SPLINE
SPL {X  -136.508, Y  +299.059, Z    +0.000, E1  +318.212, E3 -183209.129}
SPL {X  -153.176, Y  +336.305, Z    +0.000, E1  +330.872, E3 -183235.694}
SPL {X  -158.263, Y  +359.056, Z    +0.000, E1  +342.551, E3 -183242.369}
SPL {X  -159.616, Y  +371.564, Z    +0.000, E1  +350.434, E3 -183244.274}
SPL {X  -159.983, Y  +381.031, Z    +0.000, E1  +357.053, E3 -183244.964}
SPL {X  -159.990, Y  +384.524, Z    +0.000, E1  +359.995, E3 -183245.052}
SPL {X  -159.990, Y  +386.890, Z    +0.000, E1  +362.742, E3 -183245.108}
SPL {X  -159.990, Y  +392.248, Z    +0.000, E1  +370.895, E3 -183245.436}
SPL {X  -159.990, Y  +398.030, Z    +0.000, E1  +380.706, E3 -183246.087}
SPL {X  -159.990, Y  +404.858, Z    +0.000, E1  +391.125, E3 -183247.331}
SPL {X  -159.990, Y  +416.328, Z    +0.000, E1  +404.105, E3 -183250.268}
SPL {X  -159.990, Y  +459.824, Z    +0.000, E1  +420.326, E3 -183270.190}
SPL {X  -159.990, Y  +565.974, Z    +0.000, E1  +423.959, E3 -183353.679}
SPL {X  -159.990, Y  +578.588, Z    +0.000, E1  +423.918, E3 -183366.858}
SPL {X  -159.990, Y  +590.041, Z    +0.000, E1  +423.939, E3 -183378.713}
SPL {X  -159.990, Y  +601.352, Z    +0.000, E1  +423.918, E3 -183390.500}
SPL {X  -159.990, Y  +610.973, Z    +0.000, E1  +423.927, E3 -183400.468}
SPL {X  -159.990, Y  +624.756, Z    +0.000, E1  +423.949, E3 -183414.746}
SPL {X  -159.990, Y  +640.674, Z    +0.000, E1  +423.943, E3 -183431.282}
SPL {X  -159.990, Y  +652.355, Z    +0.000, E1  +423.915, E3 -183443.481}
SPL {X  -159.990, Y  +665.748, Z    +0.000, E1  +423.953, E3 -183457.335}
SPL {X  -159.643, Y  +682.032, Z    +0.000, E1  +423.894, E3 -183474.628}
SPL {X  -158.070, Y  +696.212, Z    +0.000, E1  +423.682, E3 -183490.966}
SPL {X  -155.481, Y  +709.215, Z    +0.000, E1  +423.310, E3 -183507.157}
SPL {X  -153.138, Y  +717.820, Z    +0.000, E1  +422.909, E3 -183518.576}
SPL {X  -151.229, Y  +723.716, Z    +0.000, E1  +422.630, E3 -183526.585}
SPL {X  -149.219, Y  +729.211, Z    +0.000, E1  +422.307, E3 -183534.294}
SPL {X  -146.537, Y  +735.716, Z    +0.000, E1  +421.906, E3 -183543.637}
SPL {X  -143.476, Y  +742.291, Z    +0.000, E1  +421.379, E3 -183553.397}
SPL {X  -141.015, Y  +747.074, Z    +0.000, E1  +420.958, E3 -183560.653}
SPL {X  -137.271, Y  +753.679, Z    +0.000, E1  +420.346, E3 -183570.791}
SPL {X  -133.306, Y  +759.967, Z    +0.000, E1  +419.584, E3 -183580.743}
SPL {X  -112.019, Y  +785.730, Z    +0.000, E1  +410.795, E3 -183683.484}
ENDSPLINE

SPLINE
SPL {X  -138.335, Y  +751.876, Z    +0.000, E1  +401.001, E3 -183797.783}
SPL {X  -150.285, Y  +726.376, Z    +0.000, E1  +392.667, E3 -183816.192}
SPL {X  -156.272, Y  +705.789, Z    +0.000, E1  +383.396, E3 -183823.828}
SPL {X  -159.413, Y  +685.076, Z    +0.000, E1  +371.341, E3 -183827.966}
SPL {X  -159.964, Y  +674.389, Z    +0.000, E1  +363.956, E3 -183828.937}
SPL {X  -159.990, Y  +670.214, Z    +0.000, E1  +360.653, E3 -183829.083}
SPL {X  -159.990, Y  +669.154, Z    +0.000, E1  +359.694, E3 -183829.092}
SPL {X  -159.990, Y  +666.004, Z    +0.000, E1  +355.742, E3 -183829.192}
SPL {X  -159.990, Y  +661.286, Z    +0.000, E1  +348.294, E3 -183829.508}
SPL {X  -159.990, Y  +656.470, Z    +0.000, E1  +340.220, E3 -183830.046}
SPL {X  -159.990, Y  +651.555, Z    +0.000, E1  +332.416, E3 -183830.854}
SPL {X  -159.990, Y  +640.109, Z    +0.000, E1  +318.471, E3 -183833.683}
SPL {X  -159.990, Y  +589.014, Z    +0.000, E1  +298.500, E3 -183855.548}
SPL {X  -159.990, Y  +484.717, Z    +0.000, E1  +295.169, E3 -183933.731}
SPL {X  -159.990, Y  +469.712, Z    +0.000, E1  +295.152, E3 -183948.668}
SPL {X  -159.990, Y  +456.089, Z    +0.000, E1  +295.174, E3 -183962.284}
SPL {X  -159.990, Y  +443.816, Z    +0.000, E1  +295.158, E3 -183974.484}
SPL {X  -159.990, Y  +405.035, Z    +0.000, E1  +292.209, E3 -183986.755}
SPL {X  -159.990, Y  +397.824, Z    +0.000, E1  +292.709, E3 -183997.117}
SPL {X  -159.990, Y  +393.786, Z    +0.000, E1  +293.391, E3 -184006.436}
SPL {X  -159.990, Y  +385.177, Z    +0.000, E1  +294.011, E3 -184019.553}
SPL {X  -159.935, Y  +378.300, Z    +0.000, E1  +295.100, E3 -184034.762}
SPL {X  -159.716, Y  +373.142, Z    +0.000, E1  +296.084, E3 -184047.303}
SPL {X  -158.852, Y  +363.449, Z    +0.000, E1  +296.568, E3 -184061.253}
SPL {X  -157.299, Y  +353.279, Z    +0.000, E1  +296.835, E3 -184073.685}
SPL {X  -155.242, Y  +343.812, Z    +0.000, E1  +297.102, E3 -184085.733}
SPL {X  -151.999, Y  +332.569, Z    +0.000, E1  +297.592, E3 -184100.891}
SPL {X  -148.909, Y  +323.994, Z    +0.000, E1  +298.107, E3 -184113.064}
SPL {X  -146.667, Y  +318.581, Z    +0.000, E1  +298.485, E3 -184120.985}
SPL {X  -144.416, Y  +313.647, Z    +0.000, E1  +298.845, E3 -184128.321}
SPL {X  -141.484, Y  +307.808, Z    +0.000, E1  +299.342, E3 -184137.214}
SPL {X  -139.055, Y  +303.377, Z    +0.000, E1  +299.788, E3 -184144.126}
SPL {X  -136.464, Y  +298.988, Z    +0.000, E1  +300.231, E3 -184151.001}
SPL {X  -133.486, Y  +294.305, Z    +0.000, E1  +300.785, E3 -184158.463}
SPL {X  -111.268, Y  +267.538, Z    +0.000, E1  +309.436, E3 -184266.362}
ENDSPLINE

SPLINE
SPL {X  -140.331, Y  +305.662, Z    +0.000, E1  +319.927, E3 -184378.430}
SPL {X  -153.176, Y  +336.305, Z    +0.000, E1  +330.872, E3 -184396.984}
SPL {X  -158.263, Y  +359.056, Z    +0.000, E1  +342.551, E3 -184403.659}
SPL {X  -159.616, Y  +371.564, Z    +0.000, E1  +350.434, E3 -184405.564}
SPL {X  -159.946, Y  +378.747, Z    +0.000, E1  +355.440, E3 -184406.159}
SPL {X  -159.990, Y  +384.172, Z    +0.000, E1  +359.586, E3 -184406.337}
SPL {X  -159.990, Y  +385.853, Z    +0.000, E1  +361.539, E3 -184406.362}
SPL {X  -159.990, Y  +389.234, Z    +0.000, E1  +366.142, E3 -184406.507}
SPL {X  -159.990, Y  +395.814, Z    +0.000, E1  +376.762, E3 -184407.108}
SPL {X  -159.990, Y  +404.858, Z    +0.000, E1  +391.125, E3 -184408.622}
SPL {X  -159.990, Y  +416.328, Z    +0.000, E1  +404.105, E3 -184411.559}
SPL {X  -159.990, Y  +459.824, Z    +0.000, E1  +420.326, E3 -184431.481}
SPL {X  -159.990, Y  +565.974, Z    +0.000, E1  +423.959, E3 -184514.969}
SPL {X  -159.990, Y  +578.588, Z    +0.000, E1  +423.918, E3 -184528.149}
SPL {X  -159.990, Y  +590.041, Z    +0.000, E1  +423.939, E3 -184540.004}
SPL {X  -159.990, Y  +601.352, Z    +0.000, E1  +423.918, E3 -184551.790}
SPL {X  -159.990, Y  +610.973, Z    +0.000, E1  +423.927, E3 -184561.758}
SPL {X  -159.990, Y  +624.756, Z    +0.000, E1  +423.949, E3 -184576.036}
SPL {X  -159.990, Y  +636.914, Z    +0.000, E1  +423.917, E3 -184588.712}
SPL {X  -159.990, Y  +648.849, Z    +0.000, E1  +423.945, E3 -184601.069}
SPL {X  -159.990, Y  +661.195, Z    +0.000, E1  +423.915, E3 -184613.970}
SPL {X  -159.965, Y  +674.349, Z    +0.000, E1  +423.939, E3 -184627.607}
SPL {X  -159.404, Y  +685.179, Z    +0.000, E1  +423.831, E3 -184639.486}
SPL {X  -158.535, Y  +693.032, Z    +0.000, E1  +423.713, E3 -184648.535}
SPL {X  -156.949, Y  +702.544, Z    +0.000, E1  +423.501, E3 -184660.041}
SPL {X  -154.903, Y  +711.525, Z    +0.000, E1  +423.186, E3 -184671.512}
SPL {X  -153.138, Y  +717.820, Z    +0.000, E1  +422.909, E3 -184679.866}
SPL {X  -151.229, Y  +723.716, Z    +0.000, E1  +422.630, E3 -184687.876}
SPL {X  -149.219, Y  +729.211, Z    +0.000, E1  +422.307, E3 -184695.584}
SPL {X  -146.537, Y  +735.716, Z    +0.000, E1  +421.906, E3 -184704.927}
SPL {X  -143.476, Y  +742.291, Z    +0.000, E1  +421.379, E3 -184714.687}
SPL {X  -141.015, Y  +747.074, Z    +0.000, E1  +420.958, E3 -184721.943}
SPL {X  -137.271, Y  +753.679, Z    +0.000, E1  +420.346, E3 -184732.082}
SPL {X  -133.306, Y  +759.967, Z    +0.000, E1  +419.584, E3 -184742.033}
SPL {X  -112.019, Y  +785.730, Z    +0.000, E1  +410.795, E3 -184844.774}
ENDSPLINE

SPLINE
SPL {X  -138.335, Y  +751.876, Z    +0.000, E1  +401.001, E3 -184959.073}
SPL {X  -150.285, Y  +726.376, Z    +0.000, E1  +392.667, E3 -184977.482}
SPL {X  -156.272, Y  +705.789, Z    +0.000, E1  +383.396, E3 -184985.118}
SPL {X  -159.413, Y  +685.076, Z    +0.000, E1  +371.341, E3 -184989.257}
SPL {X  -159.964, Y  +674.389, Z    +0.000, E1  +363.956, E3 -184990.227}
SPL {X  -159.990, Y  +669.409, Z    +0.000, E1  +360.015, E3 -184990.381}
SPL {X  -159.990, Y  +667.272, Z    +0.000, E1  +357.329, E3 -184990.424}
SPL {X  -159.990, Y  +664.817, Z    +0.000, E1  +353.836, E3 -184990.537}
SPL {X  -159.990, Y  +661.286, Z    +0.000, E1  +348.294, E3 -184990.799}
SPL {X  -159.990, Y  +654.198, Z    +0.000, E1  +336.753, E3 -184991.710}
SPL {X  -159.990, Y  +640.109, Z    +0.000, E1  +318.471, E3 -184994.973}
SPL {X  -159.990, Y  +589.014, Z    +0.000, E1  +298.500, E3 -185016.838}
SPL {X  -159.990, Y  +484.717, Z    +0.000, E1  +295.169, E3 -185095.022}
SPL {X  -159.990, Y  +474.300, Z    +0.000, E1  +295.184, E3 -185105.449}
SPL {X  -159.990, Y  +465.825, Z    +0.000, E1  +295.182, E3 -185113.889}
SPL {X  -159.990, Y  +451.559, Z    +0.000, E1  +295.138, E3 -185128.026}
SPL {X  -159.990, Y  +438.393, Z    +0.000, E1  +295.184, E3 -185141.248}
SPL {X  -159.990, Y  +405.035, Z    +0.000, E1  +292.209, E3 -185148.045}
SPL {X  -159.990, Y  +395.217, Z    +0.000, E1  +293.078, E3 -185164.154}
SPL {X  -159.990, Y  +387.038, Z    +0.000, E1  +293.844, E3 -185177.582}
SPL {X  -159.983, Y  +380.995, Z    +0.000, E1  +294.559, E3 -185189.151}
SPL {X  -159.795, Y  +374.602, Z    +0.000, E1  +295.796, E3 -185205.170}
SPL {X  -158.852, Y  +363.449, Z    +0.000, E1  +296.568, E3 -185222.543}
SPL {X  -156.653, Y  +349.995, Z    +0.000, E1  +296.892, E3 -185239.047}
SPL {X  -153.792, Y  +338.401, Z    +0.000, E1  +297.323, E3 -185254.216}
SPL {X  -151.244, Y  +330.327, Z    +0.000, E1  +297.748, E3 -185265.369}
SPL {X  -148.909, Y  +323.994, Z    +0.000, E1  +298.107, E3 -185274.355}
SPL {X  -146.667, Y  +318.581, Z    +0.000, E1  +298.485, E3 -185282.275}
SPL {X  -144.416, Y  +313.647, Z    +0.000, E1  +298.845, E3 -185289.611}
SPL {X  -141.484, Y  +307.808, Z    +0.000, E1  +299.342, E3 -185298.504}
SPL {X  -139.055, Y  +303.377, Z    +0.000, E1  +299.788, E3 -185305.417}
SPL {X  -136.464, Y  +298.988, Z    +0.000, E1  +300.231, E3 -185312.291}
SPL {X  -133.486, Y  +294.305, Z    +0.000, E1  +300.785, E3 -185319.753}
SPL {X  -111.268, Y  +267.538, Z    +0.000, E1  +309.436, E3 -185427.652}
ENDSPLINE

SPLINE
SPL {X  -140.331, Y  +305.662, Z    +0.000, E1  +319.927, E3 -185539.720}
SPL {X  -153.176, Y  +336.305, Z    +0.000, E1  +330.872, E3 -185558.275}
SPL {X  -157.724, Y  +355.668, Z    +0.000, E1  +340.639, E3 -185564.283}
SPL {X  -159.465, Y  +369.545, Z    +0.000, E1  +349.053, E3 -185566.605}
SPL {X  -159.983, Y  +381.031, Z    +0.000, E1  +357.053, E3 -185567.545}
SPL {X  -159.990, Y  +384.524, Z    +0.000, E1  +359.995, E3 -185567.633}
SPL {X  -159.990, Y  +386.890, Z    +0.000, E1  +362.742, E3 -185567.689}
SPL {X  -159.990, Y  +392.248, Z    +0.000, E1  +370.895, E3 -185568.016}
SPL {X  -159.990, Y  +398.030, Z    +0.000, E1  +380.706, E3 -185568.668}
SPL {X  -159.990, Y  +404.858, Z    +0.000, E1  +391.125, E3 -185569.912}
SPL {X  -159.990, Y  +416.328, Z    +0.000, E1  +404.105, E3 -185572.849}
SPL {X  -159.990, Y  +459.824, Z    +0.000, E1  +420.326, E3 -185592.771}
SPL {X  -159.990, Y  +565.974, Z    +0.000, E1  +423.959, E3 -185676.260}
SPL {X  -159.990, Y  +578.588, Z    +0.000, E1  +423.918, E3 -185689.439}
SPL {X  -159.990, Y  +590.041, Z    +0.000, E1  +423.939, E3 -185701.294}
SPL {X  -159.990, Y  +601.352, Z    +0.000, E1  +423.918, E3 -185713.080}
SPL {X  -159.990, Y  +614.998, Z    +0.000, E1  +423.962, E3 -185727.165}
SPL {X  -159.990, Y  +628.256, Z    +0.000, E1  +423.919, E3 -185741.014}
SPL {X  -159.990, Y  +640.674, Z    +0.000, E1  +423.943, E3 -185753.863}
SPL {X  -159.990, Y  +657.298, Z    +0.000, E1  +423.953, E3 -185771.135}
SPL {X  -159.990, Y  +670.369, Z    +0.000, E1  +423.912, E3 -185784.793}
SPL {X  -159.643, Y  +682.032, Z    +0.000, E1  +423.894, E3 -185797.208}
SPL {X  -158.070, Y  +696.212, Z    +0.000, E1  +423.682, E3 -185813.547}
SPL {X  -155.481, Y  +709.215, Z    +0.000, E1  +423.310, E3 -185829.738}
SPL {X  -153.138, Y  +717.820, Z    +0.000, E1  +422.909, E3 -185841.156}
SPL {X  -151.229, Y  +723.716, Z    +0.000, E1  +422.630, E3 -185849.166}
SPL {X  -149.219, Y  +729.211, Z    +0.000, E1  +422.307, E3 -185856.874}
SPL {X  -146.537, Y  +735.716, Z    +0.000, E1  +421.906, E3 -185866.217}
SPL {X  -143.476, Y  +742.291, Z    +0.000, E1  +421.379, E3 -185875.977}
SPL {X  -141.015, Y  +747.074, Z    +0.000, E1  +420.958, E3 -185883.234}
SPL {X  -137.271, Y  +753.679, Z    +0.000, E1  +420.346, E3 -185893.372}
SPL {X  -133.306, Y  +759.967, Z    +0.000, E1  +419.584, E3 -185903.324}
SPL {X  -112.019, Y  +785.730, Z    +0.000, E1  +410.795, E3 -186006.065}
ENDSPLINE

SPLINE
SPL {X  -126.527, Y  +769.417, Z    +0.000, E1  +405.012, E3 -186095.917}
SPL {X  -141.954, Y  +745.296, Z    +0.000, E1  +399.179, E3 -186127.115}
SPL {X  -153.384, Y  +716.997, Z    +0.000, E1  +388.774, E3 -186142.735}
SPL {X  -158.303, Y  +694.673, Z    +0.000, E1  +377.238, E3 -186149.046}
SPL {X  -159.604, Y  +682.609, Z    +0.000, E1  +369.664, E3 -186150.856}
SPL {X  -159.964, Y  +674.389, Z    +0.000, E1  +363.956, E3 -186151.518}
SPL {X  -159.990, Y  +669.409, Z    +0.000, E1  +360.015, E3 -186151.671}
SPL {X  -159.990, Y  +666.004, Z    +0.000, E1  +355.742, E3 -186151.773}
SPL {X  -159.990, Y  +661.286, Z    +0.000, E1  +348.294, E3 -186152.089}
SPL {X  -159.990, Y  +654.198, Z    +0.000, E1  +336.753, E3 -186153.000}
SPL {X  -159.990, Y  +640.109, Z    +0.000, E1  +318.471, E3 -186156.263}
SPL {X  -159.990, Y  +589.014, Z    +0.000, E1  +298.500, E3 -186178.129}
SPL {X  -159.990, Y  +484.717, Z    +0.000, E1  +295.169, E3 -186256.312}
SPL {X  -159.990, Y  +474.300, Z    +0.000, E1  +295.184, E3 -186266.740}
SPL {X  -159.990, Y  +465.825, Z    +0.000, E1  +295.182, E3 -186275.179}
SPL {X  -159.990, Y  +451.559, Z    +0.000, E1  +295.138, E3 -186289.316}
SPL {X  -159.990, Y  +423.512, Z    +0.000, E1  +293.559, E3 -186303.750}
SPL {X  -159.990, Y  +399.563, Z    +0.000, E1  +292.427, E3 -186316.028}
SPL {X  -159.990, Y  +393.786, Z    +0.000, E1  +293.391, E3 -186329.017}
SPL {X  -159.990, Y  +387.038, Z    +0.000, E1  +293.844, E3 -186338.873}
SPL {X  -159.983, Y  +380.995, Z    +0.000, E1  +294.559, E3 -186350.441}
SPL {X  -159.898, Y  +377.064, Z    +0.000, E1  +295.481, E3 -186361.255}
SPL {X  -159.716, Y  +373.142, Z    +0.000, E1  +296.084, E3 -186369.884}
SPL {X  -158.852, Y  +363.449, Z    +0.000, E1  +296.568, E3 -186383.834}
SPL {X  -157.299, Y  +353.279, Z    +0.000, E1  +296.835, E3 -186396.265}
SPL {X  -155.242, Y  +343.812, Z    +0.000, E1  +297.102, E3 -186408.313}
SPL {X  -151.999, Y  +332.569, Z    +0.000, E1  +297.592, E3 -186423.472}
SPL {X  -148.909, Y  +323.994, Z    +0.000, E1  +298.107, E3 -186435.645}
SPL {X  -146.667, Y  +318.581, Z    +0.000, E1  +298.485, E3 -186443.565}
SPL {X  -144.416, Y  +313.647, Z    +0.000, E1  +298.845, E3 -186450.902}
SPL {X  -141.484, Y  +307.808, Z    +0.000, E1  +299.342, E3 -186459.795}
SPL {X  -139.055, Y  +303.377, Z    +0.000, E1  +299.788, E3 -186466.707}
SPL {X  -136.464, Y  +298.988, Z    +0.000, E1  +300.231, E3 -186473.581}
SPL {X  -133.486, Y  +294.305, Z    +0.000, E1  +300.785, E3 -186481.043}
SPL {X  -111.268, Y  +267.538, Z    +0.000, E1  +309.436, E3 -186588.942}
ENDSPLINE

SPLINE
SPL {X  -140.331, Y  +305.662, Z    +0.000, E1  +319.927, E3 -186701.011}
SPL {X  -153.176, Y  +336.305, Z    +0.000, E1  +330.872, E3 -186719.565}
SPL {X  -158.263, Y  +359.056, Z    +0.000, E1  +342.551, E3 -186726.240}
SPL {X  -159.616, Y  +371.564, Z    +0.000, E1  +350.434, E3 -186728.145}
SPL {X  -159.983, Y  +381.031, Z    +0.000, E1  +357.053, E3 -186728.835}
SPL {X  -159.990, Y  +385.049, Z    +0.000, E1  +360.437, E3 -186728.931}
SPL {X  -159.990, Y  +389.234, Z    +0.000, E1  +366.142, E3 -186729.087}
SPL {X  -159.990, Y  +395.814, Z    +0.000, E1  +376.762, E3 -186729.689}
SPL {X  -159.990, Y  +404.858, Z    +0.000, E1  +391.125, E3 -186731.202}
SPL {X  -159.990, Y  +416.328, Z    +0.000, E1  +404.105, E3 -186734.139}
SPL {X  -159.990, Y  +459.824, Z    +0.000, E1  +420.326, E3 -186754.061}
SPL {X  -159.990, Y  +565.974, Z    +0.000, E1  +423.959, E3 -186837.550}
SPL {X  -159.990, Y  +582.903, Z    +0.000, E1  +423.951, E3 -186855.147}
SPL {X  -159.990, Y  +598.374, Z    +0.000, E1  +423.941, E3 -186871.234}
SPL {X  -159.990, Y  +614.998, Z    +0.000, E1  +423.962, E3 -186888.455}
SPL {X  -159.990, Y  +632.576, Z    +0.000, E1  +423.953, E3 -186906.721}
SPL {X  -159.990, Y  +648.849, Z    +0.000, E1  +423.945, E3 -186923.650}
SPL {X  -159.990, Y  +665.748, Z    +0.000, E1  +423.953, E3 -186941.206}
SPL {X  -159.643, Y  +682.032, Z    +0.000, E1  +423.894, E3 -186958.499}
SPL {X  -158.070, Y  +696.212, Z    +0.000, E1  +423.682, E3 -186974.837}
SPL {X  -155.481, Y  +709.215, Z    +0.000, E1  +423.310, E3 -186991.028}
SPL {X  -153.138, Y  +717.820, Z    +0.000, E1  +422.909, E3 -187002.447}
SPL {X  -151.229, Y  +723.716, Z    +0.000, E1  +422.630, E3 -187010.456}
SPL {X  -148.422, Y  +731.231, Z    +0.000, E1  +422.207, E3 -187021.014}
SPL {X  -145.802, Y  +737.367, Z    +0.000, E1  +421.758, E3 -187029.967}
SPL {X  -143.476, Y  +742.291, Z    +0.000, E1  +421.379, E3 -187037.268}
SPL {X  -141.015, Y  +747.074, Z    +0.000, E1  +420.958, E3 -187044.524}
SPL {X  -138.539, Y  +751.523, Z    +0.000, E1  +420.526, E3 -187051.359}
SPL {X  -136.299, Y  +755.281, Z    +0.000, E1  +420.128, E3 -187057.220}
SPL {X  -133.306, Y  +759.967, Z    +0.000, E1  +419.584, E3 -187064.614}
SPL {X  -112.019, Y  +785.730, Z    +0.000, E1  +410.795, E3 -187167.355}
ENDSPLINE

SPLINE
SPL {X  -126.527, Y  +769.417, Z    +0.000, E1  +405.012, E3 -187257.207}
SPL {X  -141.954, Y  +745.296, Z    +0.000, E1  +399.179, E3 -187288.405}
SPL {X  -153.384, Y  +716.997, Z    +0.000, E1  +388.774, E3 -187304.025}
SPL {X  -158.303, Y  +694.673, Z    +0.000, E1  +377.238, E3 -187310.337}
SPL {X  -159.604, Y  +682.609, Z    +0.000, E1  +369.664, E3 -187312.146}
SPL {X  -159.964, Y  +674.389, Z    +0.000, E1  +363.956, E3 -187312.808}
SPL {X  -159.990, Y  +669.409, Z    +0.000, E1  +360.015, E3 -187312.961}
SPL {X  -159.990, Y  +666.004, Z    +0.000, E1  +355.742, E3 -187313.063}
SPL {X  -159.990, Y  +661.286, Z    +0.000, E1  +348.294, E3 -187313.379}
SPL {X  -159.990, Y  +654.198, Z    +0.000, E1  +336.753, E3 -187314.290}
SPL {X  -159.990, Y  +640.109, Z    +0.000, E1  +318.471, E3 -187317.554}
SPL {X  -159.990, Y  +589.014, Z    +0.000, E1  +298.500, E3 -187339.419}
SPL {X  -159.990, Y  +484.717, Z    +0.000, E1  +295.169, E3 -187417.602}
SPL {X  -159.990, Y  +469.712, Z    +0.000, E1  +295.152, E3 -187432.539}
SPL {X  -159.990, Y  +456.089, Z    +0.000, E1  +295.174, E3 -187446.155}
SPL {X  -159.990, Y  +443.816, Z    +0.000, E1  +295.158, E3 -187458.355}
SPL {X  -159.990, Y  +410.689, Z    +0.000, E1  +292.263, E3 -187466.080}
SPL {X  -159.990, Y  +399.563, Z    +0.000, E1  +292.427, E3 -187477.319}
SPL {X  -159.990, Y  +393.786, Z    +0.000, E1  +293.391, E3 -187490.307}
SPL {X  -159.990, Y  +387.038, Z    +0.000, E1  +293.844, E3 -187500.163}
SPL {X  -159.983, Y  +380.995, Z    +0.000, E1  +294.559, E3 -187511.731}
SPL {X  -159.795, Y  +374.602, Z    +0.000, E1  +295.796, E3 -187527.751}
SPL {X  -159.306, Y  +367.719, Z    +0.000, E1  +296.544, E3 -187540.208}
SPL {X  -158.431, Y  +360.219, Z    +0.000, E1  +296.670, E3 -187549.059}
SPL {X  -157.299, Y  +353.279, Z    +0.000, E1  +296.835, E3 -187557.556}
SPL {X  -156.006, Y  +347.018, Z    +0.000, E1  +297.028, E3 -187565.511}
SPL {X  -153.792, Y  +338.401, Z    +0.000, E1  +297.323, E3 -187576.797}
SPL {X  -151.244, Y  +330.327, Z    +0.000, E1  +297.748, E3 -187587.950}
SPL {X  -148.909, Y  +323.994, Z    +0.000, E1  +298.107, E3 -187596.935}
SPL {X  -146.667, Y  +318.581, Z    +0.000, E1  +298.485, E3 -187604.856}
SPL {X  -144.416, Y  +313.647, Z    +0.000, E1  +298.845, E3 -187612.192}
SPL {X  -141.484, Y  +307.808, Z    +0.000, E1  +299.342, E3 -187621.085}
SPL {X  -139.055, Y  +303.377, Z    +0.000, E1  +299.788, E3 -187627.997}
SPL {X  -136.464, Y  +298.988, Z    +0.000, E1  +300.231, E3 -187634.872}
SPL {X  -133.486, Y  +294.305, Z    +0.000, E1  +300.785, E3 -187642.334}
SPL {X  -111.268, Y  +267.538, Z    +0.000, E1  +309.436, E3 -187750.233}
ENDSPLINE

SPLINE
SPL {X  -140.331, Y  +305.662, Z    +0.000, E1  +319.927, E3 -187862.301}
SPL {X  -153.176, Y  +336.305, Z    +0.000, E1  +330.872, E3 -187880.855}
SPL {X  -158.263, Y  +359.056, Z    +0.000, E1  +342.551, E3 -187887.530}
SPL {X  -159.616, Y  +371.564, Z    +0.000, E1  +350.434, E3 -187889.435}
SPL {X  -159.983, Y  +381.031, Z    +0.000, E1  +357.053, E3 -187890.125}
SPL {X  -159.990, Y  +385.049, Z    +0.000, E1  +360.437, E3 -187890.221}
SPL {X  -159.990, Y  +389.234, Z    +0.000, E1  +366.142, E3 -187890.378}
SPL {X  -159.990, Y  +395.814, Z    +0.000, E1  +376.762, E3 -187890.979}
SPL {X  -159.990, Y  +404.858, Z    +0.000, E1  +391.125, E3 -187892.493}
SPL {X  -159.990, Y  +416.328, Z    +0.000, E1  +404.105, E3 -187895.430}
SPL {X  -159.990, Y  +459.824, Z    +0.000, E1  +420.326, E3 -187915.352}
SPL {X  -159.990, Y  +565.974, Z    +0.000, E1  +423.959, E3 -187998.840}
SPL {X  -159.990, Y  +578.588, Z    +0.000, E1  +423.918, E3 -188012.020}
SPL {X  -159.990, Y  +590.041, Z    +0.000, E1  +423.939, E3 -188023.875}
SPL {X  -159.990, Y  +601.352, Z    +0.000, E1  +423.918, E3 -188035.661}
SPL {X  -159.990, Y  +610.973, Z    +0.000, E1  +423.927, E3 -188045.629}
SPL {X  -159.990, Y  +624.756, Z    +0.000, E1  +423.949, E3 -188059.907}
SPL {X  -159.990, Y  +636.914, Z    +0.000, E1  +423.917, E3 -188072.583}
SPL {X  -159.990, Y  +648.849, Z    +0.000, E1  +423.945, E3 -188084.940}
SPL {X  -159.990, Y  +661.195, Z    +0.000, E1  +423.915, E3 -188097.841}
SPL {X  -159.965, Y  +674.349, Z    +0.000, E1  +423.939, E3 -188111.478}
SPL {X  -159.404, Y  +685.179, Z    +0.000, E1  +423.831, E3 -188123.357}
SPL {X  -158.535, Y  +693.032, Z    +0.000, E1  +423.713, E3 -188132.406}
SPL {X  -156.949, Y  +702.544, Z    +0.000, E1  +423.501, E3 -188143.912}
SPL {X  -154.903, Y  +711.525, Z    +0.000, E1  +423.186, E3 -188155.383}
SPL {X  -153.138, Y  +717.820, Z    +0.000, E1  +422.909, E3 -188163.737}
SPL {X  -151.229, Y  +723.716, Z    +0.000, E1  +422.630, E3 -188171.747}
SPL {X  -148.422, Y  +731.231, Z    +0.000, E1  +422.207, E3 -188182.304}
SPL {X  -145.802, Y  +737.367, Z    +0.000, E1  +421.758, E3 -188191.257}
SPL {X  -143.476, Y  +742.291, Z    +0.000, E1  +421.379, E3 -188198.558}
SPL {X  -141.015, Y  +747.074, Z    +0.000, E1  +420.958, E3 -188205.814}
SPL {X  -137.271, Y  +753.679, Z    +0.000, E1  +420.346, E3 -188215.953}
SPL {X  -133.306, Y  +759.967, Z    +0.000, E1  +419.584, E3 -188225.904}
SPL {X  -112.019, Y  +785.730, Z    +0.000, E1  +410.795, E3 -188328.645}
ENDSPLINE

SPLINE
SPL {X  -138.335, Y  +751.876, Z    +0.000, E1  +401.001, E3 -188442.944}
SPL {X  -150.285, Y  +726.376, Z    +0.000, E1  +392.667, E3 -188461.353}
SPL {X  -154.601, Y  +712.673, Z    +0.000, E1  +386.751, E3 -188466.958}
SPL {X  -158.303, Y  +694.673, Z    +0.000, E1  +377.238, E3 -188471.627}
SPL {X  -159.774, Y  +679.819, Z    +0.000, E1  +367.840, E3 -188473.701}
SPL {X  -159.990, Y  +671.106, Z    +0.000, E1  +361.459, E3 -188474.222}
SPL {X  -159.990, Y  +669.154, Z    +0.000, E1  +359.694, E3 -188474.254}
SPL {X  -159.990, Y  +666.004, Z    +0.000, E1  +355.742, E3 -188474.353}
SPL {X  -159.990, Y  +661.286, Z    +0.000, E1  +348.294, E3 -188474.670}
SPL {X  -159.990, Y  +654.198, Z    +0.000, E1  +336.753, E3 -188475.581}
SPL {X  -159.990, Y  +640.109, Z    +0.000, E1  +318.471, E3 -188478.844}
SPL {X  -159.990, Y  +589.014, Z    +0.000, E1  +298.500, E3 -188500.709}
SPL {X  -159.990, Y  +484.717, Z    +0.000, E1  +295.169, E3 -188578.893}
SPL {X  -159.990, Y  +469.712, Z    +0.000, E1  +295.152, E3 -188593.830}
SPL {X  -159.990, Y  +456.089, Z    +0.000, E1  +295.174, E3 -188607.445}
SPL {X  -159.990, Y  +443.816, Z    +0.000, E1  +295.158, E3 -188619.646}
SPL {X  -159.990, Y  +405.035, Z    +0.000, E1  +292.209, E3 -188631.916}
SPL {X  -159.990, Y  +395.217, Z    +0.000, E1  +293.078, E3 -188648.025}
SPL {X  -159.990, Y  +385.177, Z    +0.000, E1  +294.011, E3 -188664.714}
SPL {X  -159.935, Y  +378.300, Z    +0.000, E1  +295.100, E3 -188679.924}
SPL {X  -159.533, Y  +370.414, Z    +0.000, E1  +296.253, E3 -188696.833}
SPL {X  -158.431, Y  +360.219, Z    +0.000, E1  +296.670, E3 -188710.349}
SPL {X  -157.299, Y  +353.279, Z    +0.000, E1  +296.835, E3 -188718.846}
SPL {X  -155.242, Y  +343.812, Z    +0.000, E1  +297.102, E3 -188730.894}
SPL {X  -151.999, Y  +332.569, Z    +0.000, E1  +297.592, E3 -188746.052}
SPL {X  -148.909, Y  +323.994, Z    +0.000, E1  +298.107, E3 -188758.226}
SPL {X  -146.667, Y  +318.581, Z    +0.000, E1  +298.485, E3 -188766.146}
SPL {X  -144.416, Y  +313.647, Z    +0.000, E1  +298.845, E3 -188773.482}
SPL {X  -141.484, Y  +307.808, Z    +0.000, E1  +299.342, E3 -188782.375}
SPL {X  -139.055, Y  +303.377, Z    +0.000, E1  +299.788, E3 -188789.288}
SPL {X  -136.464, Y  +298.988, Z    +0.000, E1  +300.231, E3 -188796.162}
SPL {X  -133.486, Y  +294.305, Z    +0.000, E1  +300.785, E3 -188803.624}
SPL {X  -111.268, Y  +267.538, Z    +0.000, E1  +309.436, E3 -188911.523}
ENDSPLINE

SPLINE
SPL {X  -140.331, Y  +305.662, Z    +0.000, E1  +319.927, E3 -189023.591}
SPL {X  -153.176, Y  +336.305, Z    +0.000, E1  +330.872, E3 -189042.146}
SPL {X  -157.724, Y  +355.668, Z    +0.000, E1  +340.639, E3 -189048.154}
SPL {X  -159.465, Y  +369.545, Z    +0.000, E1  +349.053, E3 -189050.476}
SPL {X  -159.983, Y  +381.031, Z    +0.000, E1  +357.053, E3 -189051.416}
SPL {X  -159.990, Y  +384.524, Z    +0.000, E1  +359.995, E3 -189051.504}
SPL {X  -159.990, Y  +385.853, Z    +0.000, E1  +361.539, E3 -189051.523}
SPL {X  -159.990, Y  +389.234, Z    +0.000, E1  +366.142, E3 -189051.668}
SPL {X  -159.990, Y  +395.814, Z    +0.000, E1  +376.762, E3 -189052.269}
SPL {X  -159.990, Y  +404.858, Z    +0.000, E1  +391.125, E3 -189053.783}
SPL {X  -159.990, Y  +416.328, Z    +0.000, E1  +404.105, E3 -189056.720}
SPL {X  -159.990, Y  +459.824, Z    +0.000, E1  +420.326, E3 -189076.642}
SPL {X  -159.990, Y  +561.459, Z    +0.000, E1  +423.923, E3 -189155.508}
SPL {X  -159.990, Y  +574.787, Z    +0.000, E1  +423.950, E3 -189169.305}
SPL {X  -159.990, Y  +590.041, Z    +0.000, E1  +423.939, E3 -189185.165}
SPL {X  -159.990, Y  +601.352, Z    +0.000, E1  +423.918, E3 -189196.951}
SPL {X  -159.990, Y  +614.998, Z    +0.000, E1  +423.962, E3 -189211.036}
SPL {X  -159.990, Y  +628.256, Z    +0.000, E1  +423.919, E3 -189224.885}
SPL {X  -159.990, Y  +640.674, Z    +0.000, E1  +423.943, E3 -189237.734}
SPL {X  -159.990, Y  +657.298, Z    +0.000, E1  +423.953, E3 -189255.006}
SPL {X  -159.990, Y  +670.369, Z    +0.000, E1  +423.912, E3 -189268.664}
SPL {X  -159.643, Y  +682.032, Z    +0.000, E1  +423.894, E3 -189281.079}
SPL {X  -158.535, Y  +693.032, Z    +0.000, E1  +423.713, E3 -189293.697}
SPL {X  -156.949, Y  +702.544, Z    +0.000, E1  +423.501, E3 -189305.202}
SPL {X  -154.903, Y  +711.525, Z    +0.000, E1  +423.186, E3 -189316.673}
SPL {X  -153.138, Y  +717.820, Z    +0.000, E1  +422.909, E3 -189325.027}
SPL {X  -151.229, Y  +723.716, Z    +0.000, E1  +422.630, E3 -189333.037}
SPL {X  -149.219, Y  +729.211, Z    +0.000, E1  +422.307, E3 -189340.745}
SPL {X  -146.537, Y  +735.716, Z    +0.000, E1  +421.906, E3 -189350.088}
SPL {X  -143.476, Y  +742.291, Z    +0.000, E1  +421.379, E3 -189359.848}
SPL {X  -141.015, Y  +747.074, Z    +0.000, E1  +420.958, E3 -189367.105}
SPL {X  -138.539, Y  +751.523, Z    +0.000, E1  +420.526, E3 -189373.939}
SPL {X  -136.299, Y  +755.281, Z    +0.000, E1  +420.128, E3 -189379.801}
SPL {X  -133.306, Y  +759.967, Z    +0.000, E1  +419.584, E3 -189387.195}
SPL {X  -112.019, Y  +785.730, Z    +0.000, E1  +410.795, E3 -189489.935}
ENDSPLINE

SPLINE
SPL {X  -138.335, Y  +751.876, Z    +0.000, E1  +401.001, E3 -189604.234}
SPL {X  -150.285, Y  +726.376, Z    +0.000, E1  +392.667, E3 -189622.643}
SPL {X  -154.601, Y  +712.673, Z    +0.000, E1  +386.751, E3 -189628.248}
SPL {X  -158.303, Y  +694.673, Z    +0.000, E1  +377.238, E3 -189632.917}
SPL {X  -159.774, Y  +679.819, Z    +0.000, E1  +367.840, E3 -189634.992}
SPL {X  -159.990, Y  +671.106, Z    +0.000, E1  +361.459, E3 -189635.512}
SPL {X  -159.990, Y  +669.154, Z    +0.000, E1  +359.694, E3 -189635.544}
SPL {X  -159.990, Y  +666.004, Z    +0.000, E1  +355.742, E3 -189635.644}
SPL {X  -159.990, Y  +661.286, Z    +0.000, E1  +348.294, E3 -189635.960}
SPL {X  -159.990, Y  +654.198, Z    +0.000, E1  +336.753, E3 -189636.871}
SPL {X  -159.990, Y  +640.109, Z    +0.000, E1  +318.471, E3 -189640.134}
SPL {X  -159.990, Y  +589.014, Z    +0.000, E1  +298.500, E3 -189662.000}
SPL {X  -159.990, Y  +484.717, Z    +0.000, E1  +295.169, E3 -189740.183}
SPL {X  -159.990, Y  +474.300, Z    +0.000, E1  +295.184, E3 -189750.611}
SPL {X  -159.990, Y  +465.825, Z    +0.000, E1  +295.182, E3 -189759.050}
SPL {X  -159.990, Y  +451.559, Z    +0.000, E1  +295.138, E3 -189773.187}
SPL {X  -159.990, Y  +423.512, Z    +0.000, E1  +293.559, E3 -189787.621}
SPL {X  -159.990, Y  +399.563, Z    +0.000, E1  +292.427, E3 -189799.899}
SPL {X  -159.990, Y  +393.786, Z    +0.000, E1  +293.391, E3 -189812.888}
SPL {X  -159.990, Y  +387.038, Z    +0.000, E1  +293.844, E3 -189822.744}
SPL {X  -159.983, Y  +380.995, Z    +0.000, E1  +294.559, E3 -189834.312}
SPL {X  -159.898, Y  +377.064, Z    +0.000, E1  +295.481, E3 -189845.126}
SPL {X  -159.533, Y  +370.414, Z    +0.000, E1  +296.253, E3 -189858.123}
SPL {X  -158.431, Y  +360.219, Z    +0.000, E1  +296.670, E3 -189871.640}
SPL {X  -157.299, Y  +353.279, Z    +0.000, E1  +296.835, E3 -189880.136}
SPL {X  -156.006, Y  +347.018, Z    +0.000, E1  +297.028, E3 -189888.092}
SPL {X  -153.792, Y  +338.401, Z    +0.000, E1  +297.323, E3 -189899.378}
SPL {X  -151.244, Y  +330.327, Z    +0.000, E1  +297.748, E3 -189910.530}
SPL {X  -148.909, Y  +323.994, Z    +0.000, E1  +298.107, E3 -189919.516}
SPL {X  -146.667, Y  +318.581, Z    +0.000, E1  +298.485, E3 -189927.436}
SPL {X  -144.416, Y  +313.647, Z    +0.000, E1  +298.845, E3 -189934.773}
SPL {X  -141.484, Y  +307.808, Z    +0.000, E1  +299.342, E3 -189943.666}
SPL {X  -139.055, Y  +303.377, Z    +0.000, E1  +299.788, E3 -189950.578}
SPL {X  -136.464, Y  +298.988, Z    +0.000, E1  +300.231, E3 -189957.452}
SPL {X  -133.486, Y  +294.305, Z    +0.000, E1  +300.785, E3 -189964.914}
SPL {X  -111.268, Y  +267.538, Z    +0.000, E1  +309.436, E3 -190072.813}
ENDSPLINE

SPLINE
SPL {X  -140.331, Y  +305.662, Z    +0.000, E1  +319.927, E3 -190184.881}
SPL {X  -153.176, Y  +336.305, Z    +0.000, E1  +330.872, E3 -190203.436}
SPL {X  -158.263, Y  +359.056, Z    +0.000, E1  +342.551, E3 -190210.111}
SPL {X  -159.616, Y  +371.564, Z    +0.000, E1  +350.434, E3 -190212.016}
SPL {X  -159.983, Y  +381.031, Z    +0.000, E1  +357.053, E3 -190212.706}
SPL {X  -159.990, Y  +384.524, Z    +0.000, E1  +359.995, E3 -190212.794}
SPL {X  -159.990, Y  +386.890, Z    +0.000, E1  +362.742, E3 -190212.850}
SPL {X  -159.990, Y  +392.248, Z    +0.000, E1  +370.895, E3 -190213.178}
SPL {X  -159.990, Y  +398.030, Z    +0.000, E1  +380.706, E3 -190213.829}
SPL {X  -159.990, Y  +404.858, Z    +0.000, E1  +391.125, E3 -190215.073}
SPL {X  -159.990, Y  +416.328, Z    +0.000, E1  +404.105, E3 -190218.010}
SPL {X  -159.990, Y  +459.824, Z    +0.000, E1  +420.326, E3 -190237.932}
SPL {X  -159.990, Y  +565.974, Z    +0.000, E1  +423.959, E3 -190321.421}
SPL {X  -159.990, Y  +578.588, Z    +0.000, E1  +423.918, E3 -190334.600}
SPL {X  -159.990, Y  +590.041, Z    +0.000, E1  +423.939, E3 -190346.455}
SPL {X  -159.990, Y  +601.352, Z    +0.000, E1  +423.918, E3 -190358.242}
SPL {X  -159.990, Y  +610.973, Z    +0.000, E1  +423.927, E3 -190368.210}
SPL {X  -159.990, Y  +624.756, Z    +0.000, E1  +423.949, E3 -190382.488}
SPL {X  -159.990, Y  +640.674, Z    +0.000, E1  +423.943, E3 -190399.024}
SPL {X  -159.990, Y  +652.355, Z    +0.000, E1  +423.915, E3 -190411.223}
SPL {X  -159.990, Y  +665.748, Z    +0.000, E1  +423.953, E3 -190425.077}
SPL {X  -159.643, Y  +682.032, Z    +0.000, E1  +423.894, E3 -190442.370}
SPL {X  -158.070, Y  +696.212, Z    +0.000, E1  +423.682, E3 -190458.708}
SPL {X  -155.481, Y  +709.215, Z    +0.000, E1  +423.310, E3 -190474.899}
SPL {X  -153.138, Y  +717.820, Z    +0.000, E1  +422.909, E3 -190486.318}
SPL {X  -151.229, Y  +723.716, Z    +0.000, E1  +422.630, E3 -190494.327}
SPL {X  -148.422, Y  +731.231, Z    +0.000, E1  +422.207, E3 -190504.885}
SPL {X  -145.802, Y  +737.367, Z    +0.000, E1  +421.758, E3 -190513.838}
SPL {X  -143.476, Y  +742.291, Z    +0.000, E1  +421.379, E3 -190521.139}
SPL {X  -141.015, Y  +747.074, Z    +0.000, E1  +420.958, E3 -190528.395}
SPL {X  -138.539, Y  +751.523, Z    +0.000, E1  +420.526, E3 -190535.230}
SPL {X  -136.299, Y  +755.281, Z    +0.000, E1  +420.128, E3 -190541.091}
SPL {X  -133.306, Y  +759.967, Z    +0.000, E1  +419.584, E3 -190548.485}
SPL {X  -112.019, Y  +785.730, Z    +0.000, E1  +410.795, E3 -190651.226}
ENDSPLINE

SPLINE
SPL {X  -138.335, Y  +751.876, Z    +0.000, E1  +401.001, E3 -190765.525}
SPL {X  -150.285, Y  +726.376, Z    +0.000, E1  +392.667, E3 -190783.934}
SPL {X  -154.601, Y  +712.673, Z    +0.000, E1  +386.751, E3 -190789.539}
SPL {X  -158.303, Y  +694.673, Z    +0.000, E1  +377.238, E3 -190794.208}
SPL {X  -159.774, Y  +679.819, Z    +0.000, E1  +367.840, E3 -190796.282}
SPL {X  -159.990, Y  +671.106, Z    +0.000, E1  +361.459, E3 -190796.803}
SPL {X  -159.990, Y  +669.154, Z    +0.000, E1  +359.694, E3 -190796.834}
SPL {X  -159.990, Y  +666.004, Z    +0.000, E1  +355.742, E3 -190796.934}
SPL {X  -159.990, Y  +661.286, Z    +0.000, E1  +348.294, E3 -190797.250}
SPL {X  -159.990, Y  +656.470, Z    +0.000, E1  +340.220, E3 -190797.788}
SPL {X  -159.990, Y  +651.555, Z    +0.000, E1  +332.416, E3 -190798.596}
SPL {X  -159.990, Y  +640.109, Z    +0.000, E1  +318.471, E3 -190801.425}
SPL {X  -159.990, Y  +589.014, Z    +0.000, E1  +298.500, E3 -190823.290}
SPL {X  -159.990, Y  +484.717, Z    +0.000, E1  +295.169, E3 -190901.473}
SPL {X  -159.990, Y  +474.300, Z    +0.000, E1  +295.184, E3 -190911.901}
SPL {X  -159.990, Y  +460.248, Z    +0.000, E1  +295.138, E3 -190925.811}
SPL {X  -159.990, Y  +443.816, Z    +0.000, E1  +295.158, E3 -190942.226}
SPL {X  -159.990, Y  +410.689, Z    +0.000, E1  +292.263, E3 -190949.951}
SPL {X  -159.990, Y  +399.563, Z    +0.000, E1  +292.427, E3 -190961.190}
SPL {X  -159.990, Y  +393.786, Z    +0.000, E1  +293.391, E3 -190974.178}
SPL {X  -159.990, Y  +387.038, Z    +0.000, E1  +293.844, E3 -190984.034}
SPL {X  -159.983, Y  +380.995, Z    +0.000, E1  +294.559, E3 -190995.602}
SPL {X  -159.795, Y  +374.602, Z    +0.000, E1  +295.796, E3 -191011.622}
SPL {X  -158.852, Y  +363.449, Z    +0.000, E1  +296.568, E3 -191028.995}
SPL {X  -156.653, Y  +349.995, Z    +0.000, E1  +296.892, E3 -191045.498}
SPL {X  -153.792, Y  +338.401, Z    +0.000, E1  +297.323, E3 -191060.668}
SPL {X  -151.244, Y  +330.327, Z    +0.000, E1  +297.748, E3 -191071.821}
SPL {X  -148.909, Y  +323.994, Z    +0.000, E1  +298.107, E3 -191080.806}
SPL {X  -146.667, Y  +318.581, Z    +0.000, E1  +298.485, E3 -191088.727}
SPL {X  -144.416, Y  +313.647, Z    +0.000, E1  +298.845, E3 -191096.063}
SPL {X  -141.484, Y  +307.808, Z    +0.000, E1  +299.342, E3 -191104.956}
SPL {X  -139.055, Y  +303.377, Z    +0.000, E1  +299.788, E3 -191111.868}
SPL {X  -136.464, Y  +298.988, Z    +0.000, E1  +300.231, E3 -191118.743}
SPL {X  -133.486, Y  +294.305, Z    +0.000, E1  +300.785, E3 -191126.205}
SPL {X  -111.198, Y  +267.470, Z    +0.000, E1  +308.990, E3 -191227.225}
ENDSPLINE

SPLINE
SPL {X  -136.508, Y  +299.059, Z    +0.000, E1  +318.212, E3 -191338.161}
SPL {X  -153.176, Y  +336.305, Z    +0.000, E1  +330.872, E3 -191364.726}
SPL {X  -158.263, Y  +359.056, Z    +0.000, E1  +342.551, E3 -191371.401}
SPL {X  -159.616, Y  +371.564, Z    +0.000, E1  +350.434, E3 -191373.306}
SPL {X  -159.983, Y  +381.031, Z    +0.000, E1  +357.053, E3 -191373.996}
SPL {X  -159.990, Y  +384.524, Z    +0.000, E1  +359.995, E3 -191374.085}
SPL {X  -159.990, Y  +386.890, Z    +0.000, E1  +362.742, E3 -191374.141}
SPL {X  -159.990, Y  +392.248, Z    +0.000, E1  +370.895, E3 -191374.468}
SPL {X  -159.990, Y  +398.030, Z    +0.000, E1  +380.706, E3 -191375.119}
SPL {X  -159.990, Y  +404.858, Z    +0.000, E1  +391.125, E3 -191376.364}
SPL {X  -159.990, Y  +416.328, Z    +0.000, E1  +404.105, E3 -191379.301}
SPL {X  -159.990, Y  +459.824, Z    +0.000, E1  +420.326, E3 -191399.223}
SPL {X  -159.990, Y  +565.974, Z    +0.000, E1  +423.959, E3 -191482.711}
SPL {X  -159.990, Y  +578.588, Z    +0.000, E1  +423.918, E3 -191495.891}
SPL {X  -159.990, Y  +590.041, Z    +0.000, E1  +423.939, E3 -191507.746}
SPL {X  -159.990, Y  +601.352, Z    +0.000, E1  +423.918, E3 -191519.532}
SPL {X  -159.990, Y  +610.973, Z    +0.000, E1  +423.927, E3 -191529.500}
SPL {X  -159.990, Y  +624.756, Z    +0.000, E1  +423.949, E3 -191543.778}
SPL {X  -159.990, Y  +640.674, Z    +0.000, E1  +423.943, E3 -191560.315}
SPL {X  -159.990, Y  +657.298, Z    +0.000, E1  +423.953, E3 -191577.587}
SPL {X  -159.965, Y  +674.349, Z    +0.000, E1  +423.939, E3 -191595.349}
SPL {X  -159.404, Y  +685.179, Z    +0.000, E1  +423.831, E3 -191607.227}
SPL {X  -158.535, Y  +693.032, Z    +0.000, E1  +423.713, E3 -191616.277}
SPL {X  -156.949, Y  +702.544, Z    +0.000, E1  +423.501, E3 -191627.782}
SPL {X  -154.903, Y  +711.525, Z    +0.000, E1  +423.186, E3 -191639.253}
SPL {X  -153.138, Y  +717.820, Z    +0.000, E1  +422.909, E3 -191647.608}
SPL {X  -151.229, Y  +723.716, Z    +0.000, E1  +422.630, E3 -191655.618}
SPL {X  -148.422, Y  +731.231, Z    +0.000, E1  +422.207, E3 -191666.175}
SPL {X  -145.802, Y  +737.367, Z    +0.000, E1  +421.758, E3 -191675.128}
SPL {X  -143.476, Y  +742.291, Z    +0.000, E1  +421.379, E3 -191682.429}
SPL {X  -141.015, Y  +747.074, Z    +0.000, E1  +420.958, E3 -191689.685}
SPL {X  -137.271, Y  +753.679, Z    +0.000, E1  +420.346, E3 -191699.824}
SPL {X  -133.306, Y  +759.967, Z    +0.000, E1  +419.584, E3 -191709.775}
SPL {X  -112.019, Y  +785.730, Z    +0.000, E1  +410.795, E3 -191812.516}
ENDSPLINE

SPLINE
SPL {X  -138.335, Y  +751.876, Z    +0.000, E1  +401.001, E3 -191926.815}
SPL {X  -150.285, Y  +726.376, Z    +0.000, E1  +392.667, E3 -191945.224}
SPL {X  -154.601, Y  +712.673, Z    +0.000, E1  +386.751, E3 -191950.829}
SPL {X  -158.303, Y  +694.673, Z    +0.000, E1  +377.238, E3 -191955.498}
SPL {X  -159.774, Y  +679.819, Z    +0.000, E1  +367.840, E3 -191957.572}
SPL {X  -159.990, Y  +671.106, Z    +0.000, E1  +361.459, E3 -191958.093}
SPL {X  -159.990, Y  +669.154, Z    +0.000, E1  +359.694, E3 -191958.125}
SPL {X  -159.990, Y  +666.004, Z    +0.000, E1  +355.742, E3 -191958.224}
SPL {X  -159.990, Y  +661.286, Z    +0.000, E1  +348.294, E3 -191958.541}
SPL {X  -159.990, Y  +654.198, Z    +0.000, E1  +336.753, E3 -191959.452}
SPL {X  -159.990, Y  +640.109, Z    +0.000, E1  +318.471, E3 -191962.715}
SPL {X  -159.990, Y  +589.014, Z    +0.000, E1  +298.500, E3 -191984.580}
SPL {X  -159.990, Y  +484.717, Z    +0.000, E1  +295.169, E3 -192062.763}
SPL {X  -159.990, Y  +474.300, Z    +0.000, E1  +295.184, E3 -192073.191}
SPL {X  -159.990, Y  +460.248, Z    +0.000, E1  +295.138, E3 -192087.101}
SPL {X  -159.990, Y  +443.816, Z    +0.000, E1  +295.158, E3 -192103.517}
SPL {X  -159.990, Y  +405.035, Z    +0.000, E1  +292.209, E3 -192115.787}
SPL {X  -159.990, Y  +397.824, Z    +0.000, E1  +292.709, E3 -192126.149}
SPL {X  -159.990, Y  +393.786, Z    +0.000, E1  +293.391, E3 -192135.468}
SPL {X  -159.990, Y  +387.038, Z    +0.000, E1  +293.844, E3 -192145.324}
SPL {X  -159.983, Y  +380.995, Z    +0.000, E1  +294.559, E3 -192156.893}
SPL {X  -159.898, Y  +377.064, Z    +0.000, E1  +295.481, E3 -192167.707}
SPL {X  -159.533, Y  +370.414, Z    +0.000, E1  +296.253, E3 -192180.704}
SPL {X  -158.431, Y  +360.219, Z    +0.000, E1  +296.670, E3 -192194.220}
SPL {X  -157.299, Y  +353.279, Z    +0.000, E1  +296.835, E3 -192202.717}
SPL {X  -156.006, Y  +347.018, Z    +0.000, E1  +297.028, E3 -192210.672}
SPL {X  -153.792, Y  +338.401, Z    +0.000, E1  +297.323, E3 -192221.958}
SPL {X  -151.244, Y  +330.327, Z    +0.000, E1  +297.748, E3 -192233.111}
SPL {X  -148.909, Y  +323.994, Z    +0.000, E1  +298.107, E3 -192242.097}
SPL {X  -146.667, Y  +318.581, Z    +0.000, E1  +298.485, E3 -192250.017}
SPL {X  -144.416, Y  +313.647, Z    +0.000, E1  +298.845, E3 -192257.353}
SPL {X  -141.484, Y  +307.808, Z    +0.000, E1  +299.342, E3 -192266.246}
SPL {X  -139.055, Y  +303.377, Z    +0.000, E1  +299.788, E3 -192273.158}
SPL {X  -136.464, Y  +298.988, Z    +0.000, E1  +300.231, E3 -192280.033}
SPL {X  -133.486, Y  +294.305, Z    +0.000, E1  +300.785, E3 -192287.495}
SPL {X  -111.268, Y  +267.538, Z    +0.000, E1  +309.436, E3 -192395.394}
ENDSPLINE

SPLINE
SPL {X  -140.331, Y  +305.662, Z    +0.000, E1  +319.927, E3 -192507.462}
SPL {X  -153.176, Y  +336.305, Z    +0.000, E1  +330.872, E3 -192526.016}
SPL {X  -158.263, Y  +359.056, Z    +0.000, E1  +342.551, E3 -192532.691}
SPL {X  -159.616, Y  +371.564, Z    +0.000, E1  +350.434, E3 -192534.596}
SPL {X  -159.983, Y  +381.031, Z    +0.000, E1  +357.053, E3 -192535.287}
SPL {X  -159.990, Y  +384.524, Z    +0.000, E1  +359.995, E3 -192535.375}
SPL {X  -159.990, Y  +386.890, Z    +0.000, E1  +362.742, E3 -192535.431}
SPL {X  -159.990, Y  +392.248, Z    +0.000, E1  +370.895, E3 -192535.758}
SPL {X  -159.990, Y  +398.030, Z    +0.000, E1  +380.706, E3 -192536.410}
SPL {X  -159.990, Y  +404.858, Z    +0.000, E1  +391.125, E3 -192537.654}
SPL {X  -159.990, Y  +416.328, Z    +0.000, E1  +404.105, E3 -192540.591}
SPL {X  -159.990, Y  +459.824, Z    +0.000, E1  +420.326, E3 -192560.513}
SPL {X  -159.990, Y  +565.974, Z    +0.000, E1  +423.959, E3 -192644.002}
SPL {X  -159.990, Y  +578.588, Z    +0.000, E1  +423.918, E3 -192657.181}
SPL {X  -159.990, Y  +590.041, Z    +0.000, E1  +423.939, E3 -192669.036}
SPL {X  -159.990, Y  +601.352, Z    +0.000, E1  +423.918, E3 -192680.822}
SPL {X  -159.990, Y  +610.973, Z    +0.000, E1  +423.927, E3 -192690.790}
SPL {X  -159.990, Y  +624.756, Z    +0.000, E1  +423.949, E3 -192705.068}
SPL {X  -159.990, Y  +640.674, Z    +0.000, E1  +423.943, E3 -192721.605}
SPL {X  -159.990, Y  +652.355, Z    +0.000, E1  +423.915, E3 -192733.803}
SPL {X  -159.990, Y  +665.748, Z    +0.000, E1  +423.953, E3 -192747.657}
SPL {X  -159.643, Y  +682.032, Z    +0.000, E1  +423.894, E3 -192764.950}
SPL {X  -158.535, Y  +693.032, Z    +0.000, E1  +423.713, E3 -192777.568}
SPL {X  -156.949, Y  +702.544, Z    +0.000, E1  +423.501, E3 -192789.073}
SPL {X  -154.903, Y  +711.525, Z    +0.000, E1  +423.186, E3 -192800.544}
SPL {X  -153.138, Y  +717.820, Z    +0.000, E1  +422.909, E3 -192808.898}
SPL {X  -151.229, Y  +723.716, Z    +0.000, E1  +422.630, E3 -192816.908}
SPL {X  -148.422, Y  +731.231, Z    +0.000, E1  +422.207, E3 -192827.466}
SPL {X  -145.802, Y  +737.367, Z    +0.000, E1  +421.758, E3 -192836.419}
SPL {X  -143.476, Y  +742.291, Z    +0.000, E1  +421.379, E3 -192843.719}
SPL {X  -141.015, Y  +747.074, Z    +0.000, E1  +420.958, E3 -192850.976}
SPL {X  -137.271, Y  +753.679, Z    +0.000, E1  +420.346, E3 -192861.114}
SPL {X  -133.306, Y  +759.967, Z    +0.000, E1  +419.584, E3 -192871.066}
SPL {X  -112.019, Y  +785.730, Z    +0.000, E1  +410.795, E3 -192973.806}
ENDSPLINE

SPLINE
SPL {X  -138.335, Y  +751.876, Z    +0.000, E1  +401.001, E3 -193088.105}
SPL {X  -150.285, Y  +726.376, Z    +0.000, E1  +392.667, E3 -193106.514}
SPL {X  -154.601, Y  +712.673, Z    +0.000, E1  +386.751, E3 -193112.119}
SPL {X  -158.303, Y  +694.673, Z    +0.000, E1  +377.238, E3 -193116.788}
SPL {X  -159.774, Y  +679.819, Z    +0.000, E1  +367.840, E3 -193118.863}
SPL {X  -159.990, Y  +671.106, Z    +0.000, E1  +361.459, E3 -193119.383}
SPL {X  -159.990, Y  +669.154, Z    +0.000, E1  +359.694, E3 -193119.415}
SPL {X  -159.990, Y  +666.004, Z    +0.000, E1  +355.742, E3 -193119.515}
SPL {X  -159.990, Y  +661.286, Z    +0.000, E1  +348.294, E3 -193119.831}
SPL {X  -159.990, Y  +656.470, Z    +0.000, E1  +340.220, E3 -193120.368}
SPL {X  -159.990, Y  +651.555, Z    +0.000, E1  +332.416, E3 -193121.176}
SPL {X  -159.990, Y  +640.109, Z    +0.000, E1  +318.471, E3 -193124.005}
SPL {X  -159.990, Y  +589.014, Z    +0.000, E1  +298.500, E3 -193145.871}
SPL {X  -159.990, Y  +484.717, Z    +0.000, E1  +295.169, E3 -193224.054}
SPL {X  -159.990, Y  +474.300, Z    +0.000, E1  +295.184, E3 -193234.482}
SPL {X  -159.990, Y  +460.248, Z    +0.000, E1  +295.138, E3 -193248.392}
SPL {X  -159.990, Y  +443.816, Z    +0.000, E1  +295.158, E3 -193264.807}
SPL {X  -159.990, Y  +410.689, Z    +0.000, E1  +292.263, E3 -193272.531}
SPL {X  -159.990, Y  +399.563, Z    +0.000, E1  +292.427, E3 -193283.770}
SPL {X  -159.990, Y  +393.786, Z    +0.000, E1  +293.391, E3 -193296.759}
SPL {X  -159.990, Y  +387.038, Z    +0.000, E1  +293.844, E3 -193306.615}
SPL {X  -159.983, Y  +380.995, Z    +0.000, E1  +294.559, E3 -193318.183}
SPL {X  -159.898, Y  +377.064, Z    +0.000, E1  +295.481, E3 -193328.997}
SPL {X  -159.533, Y  +370.414, Z    +0.000, E1  +296.253, E3 -193341.994}
SPL {X  -158.431, Y  +360.219, Z    +0.000, E1  +296.670, E3 -193355.511}
SPL {X  -157.299, Y  +353.279, Z    +0.000, E1  +296.835, E3 -193364.007}
SPL {X  -155.242, Y  +343.812, Z    +0.000, E1  +297.102, E3 -193376.055}
SPL {X  -151.999, Y  +332.569, Z    +0.000, E1  +297.592, E3 -193391.214}
SPL {X  -148.909, Y  +323.994, Z    +0.000, E1  +298.107, E3 -193403.387}
SPL {X  -146.667, Y  +318.581, Z    +0.000, E1  +298.485, E3 -193411.307}
SPL {X  -144.416, Y  +313.647, Z    +0.000, E1  +298.845, E3 -193418.644}
SPL {X  -141.484, Y  +307.808, Z    +0.000, E1  +299.342, E3 -193427.537}
SPL {X  -139.055, Y  +303.377, Z    +0.000, E1  +299.788, E3 -193434.449}
SPL {X  -136.464, Y  +298.988, Z    +0.000, E1  +300.231, E3 -193441.323}
SPL {X  -133.486, Y  +294.305, Z    +0.000, E1  +300.785, E3 -193448.785}
SPL {X  -111.268, Y  +267.538, Z    +0.000, E1  +309.436, E3 -193556.684}
ENDSPLINE

SPLINE
SPL {X  -140.331, Y  +305.662, Z    +0.000, E1  +319.927, E3 -193668.752}
SPL {X  -153.176, Y  +336.305, Z    +0.000, E1  +330.872, E3 -193687.307}
SPL {X  -157.724, Y  +355.668, Z    +0.000, E1  +340.639, E3 -193693.315}
SPL {X  -159.465, Y  +369.545, Z    +0.000, E1  +349.053, E3 -193695.637}
SPL {X  -159.983, Y  +381.031, Z    +0.000, E1  +357.053, E3 -193696.577}
SPL {X  -159.990, Y  +384.524, Z    +0.000, E1  +359.995, E3 -193696.665}
SPL {X  -159.990, Y  +385.853, Z    +0.000, E1  +361.539, E3 -193696.685}
SPL {X  -159.990, Y  +389.234, Z    +0.000, E1  +366.142, E3 -193696.829}
SPL {X  -159.990, Y  +395.814, Z    +0.000, E1  +376.762, E3 -193697.430}
SPL {X  -159.990, Y  +404.858, Z    +0.000, E1  +391.125, E3 -193698.944}
SPL {X  -159.990, Y  +416.328, Z    +0.000, E1  +404.105, E3 -193701.881}
SPL {X  -159.990, Y  +459.824, Z    +0.000, E1  +420.326, E3 -193721.803}
SPL {X  -159.990, Y  +561.459, Z    +0.000, E1  +423.923, E3 -193800.670}
SPL {X  -159.990, Y  +574.787, Z    +0.000, E1  +423.950, E3 -193814.466}
SPL {X  -159.990, Y  +590.041, Z    +0.000, E1  +423.939, E3 -193830.326}
SPL {X  -159.990, Y  +601.352, Z    +0.000, E1  +423.918, E3 -193842.113}
SPL {X  -159.990, Y  +614.998, Z    +0.000, E1  +423.962, E3 -193856.197}
SPL {X  -159.990, Y  +628.256, Z    +0.000, E1  +423.919, E3 -193870.046}
SPL {X  -159.990, Y  +640.674, Z    +0.000, E1  +423.943, E3 -193882.895}
SPL {X  -159.990, Y  +657.298, Z    +0.000, E1  +423.953, E3 -193900.167}
SPL {X  -159.990, Y  +670.369, Z    +0.000, E1  +423.912, E3 -193913.825}
SPL {X  -159.643, Y  +682.032, Z    +0.000, E1  +423.894, E3 -193926.241}
SPL {X  -158.535, Y  +693.032, Z    +0.000, E1  +423.713, E3 -193938.858}
SPL {X  -156.949, Y  +702.544, Z    +0.000, E1  +423.501, E3 -193950.363}
SPL {X  -154.903, Y  +711.525, Z    +0.000, E1  +423.186, E3 -193961.834}
SPL {X  -153.138, Y  +717.820, Z    +0.000, E1  +422.909, E3 -193970.188}
SPL {X  -151.229, Y  +723.716, Z    +0.000, E1  +422.630, E3 -193978.198}
SPL {X  -149.219, Y  +729.211, Z    +0.000, E1  +422.307, E3 -193985.906}
SPL {X  -146.537, Y  +735.716, Z    +0.000, E1  +421.906, E3 -193995.250}
SPL {X  -143.476, Y  +742.291, Z    +0.000, E1  +421.379, E3 -194005.010}
SPL {X  -141.015, Y  +747.074, Z    +0.000, E1  +420.958, E3 -194012.266}
SPL {X  -138.539, Y  +751.523, Z    +0.000, E1  +420.526, E3 -194019.101}
SPL {X  -136.299, Y  +755.281, Z    +0.000, E1  +420.128, E3 -194024.962}
SPL {X  -133.306, Y  +759.967, Z    +0.000, E1  +419.584, E3 -194032.356}
SPL {X  -112.019, Y  +785.730, Z    +0.000, E1  +410.795, E3 -194135.097}
ENDSPLINE

SPLINE
SPL {X  -138.335, Y  +751.876, Z    +0.000, E1  +401.001, E3 -194249.396}
SPL {X  -150.285, Y  +726.376, Z    +0.000, E1  +392.667, E3 -194267.805}
SPL {X  -154.601, Y  +712.673, Z    +0.000, E1  +386.751, E3 -194273.410}
SPL {X  -158.303, Y  +694.673, Z    +0.000, E1  +377.238, E3 -194278.079}
SPL {X  -159.774, Y  +679.819, Z    +0.000, E1  +367.840, E3 -194280.153}
SPL {X  -159.990, Y  +671.106, Z    +0.000, E1  +361.459, E3 -194280.674}
SPL {X  -159.990, Y  +669.154, Z    +0.000, E1  +359.694, E3 -194280.705}
SPL {X  -159.990, Y  +666.004, Z    +0.000, E1  +355.742, E3 -194280.805}
SPL {X  -159.990, Y  +661.286, Z    +0.000, E1  +348.294, E3 -194281.121}
SPL {X  -159.990, Y  +654.198, Z    +0.000, E1  +336.753, E3 -194282.032}
SPL {X  -159.990, Y  +640.109, Z    +0.000, E1  +318.471, E3 -194285.296}
SPL {X  -159.990, Y  +589.014, Z    +0.000, E1  +298.500, E3 -194307.161}
SPL {X  -159.990, Y  +484.717, Z    +0.000, E1  +295.169, E3 -194385.344}
SPL {X  -159.990, Y  +474.300, Z    +0.000, E1  +295.184, E3 -194395.772}
SPL {X  -159.990, Y  +465.825, Z    +0.000, E1  +295.182, E3 -194404.211}
SPL {X  -159.990, Y  +451.559, Z    +0.000, E1  +295.138, E3 -194418.348}
SPL {X  -159.990, Y  +438.393, Z    +0.000, E1  +295.184, E3 -194431.570}
SPL {X  -159.990, Y  +405.035, Z    +0.000, E1  +292.209, E3 -194438.368}
SPL {X  -159.990, Y  +395.217, Z    +0.000, E1  +293.078, E3 -194454.477}
SPL {X  -159.990, Y  +387.038, Z    +0.000, E1  +293.844, E3 -194467.905}
SPL {X  -159.983, Y  +380.995, Z    +0.000, E1  +294.559, E3 -194479.473}
SPL {X  -159.795, Y  +374.602, Z    +0.000, E1  +295.796, E3 -194495.493}
SPL {X  -158.852, Y  +363.449, Z    +0.000, E1  +296.568, E3 -194512.866}
SPL {X  -157.299, Y  +353.279, Z    +0.000, E1  +296.835, E3 -194525.298}
SPL {X  -155.242, Y  +343.812, Z    +0.000, E1  +297.102, E3 -194537.346}
SPL {X  -151.999, Y  +332.569, Z    +0.000, E1  +297.592, E3 -194552.504}
SPL {X  -148.909, Y  +323.994, Z    +0.000, E1  +298.107, E3 -194564.677}
SPL {X  -146.667, Y  +318.581, Z    +0.000, E1  +298.485, E3 -194572.598}
SPL {X  -144.416, Y  +313.647, Z    +0.000, E1  +298.845, E3 -194579.934}
SPL {X  -141.484, Y  +307.808, Z    +0.000, E1  +299.342, E3 -194588.827}
SPL {X  -139.055, Y  +303.377, Z    +0.000, E1  +299.788, E3 -194595.739}
SPL {X  -136.464, Y  +298.988, Z    +0.000, E1  +300.231, E3 -194602.614}
SPL {X  -133.486, Y  +294.305, Z    +0.000, E1  +300.785, E3 -194610.076}
SPL {X  -111.268, Y  +267.538, Z    +0.000, E1  +309.436, E3 -194717.975}
ENDSPLINE

SPLINE
SPL {X  -140.331, Y  +305.662, Z    +0.000, E1  +319.927, E3 -194830.043}
SPL {X  -153.176, Y  +336.305, Z    +0.000, E1  +330.872, E3 -194848.597}
SPL {X  -158.263, Y  +359.056, Z    +0.000, E1  +342.551, E3 -194855.272}
SPL {X  -159.616, Y  +371.564, Z    +0.000, E1  +350.434, E3 -194857.177}
SPL {X  -159.983, Y  +381.031, Z    +0.000, E1  +357.053, E3 -194857.867}
SPL {X  -159.990, Y  +384.524, Z    +0.000, E1  +359.995, E3 -194857.956}
SPL {X  -159.990, Y  +386.890, Z    +0.000, E1  +362.742, E3 -194858.012}
SPL {X  -159.990, Y  +392.248, Z    +0.000, E1  +370.895, E3 -194858.339}
SPL {X  -159.990, Y  +398.030, Z    +0.000, E1  +380.706, E3 -194858.990}
SPL {X  -159.990, Y  +404.858, Z    +0.000, E1  +391.125, E3 -194860.235}
SPL {X  -159.990, Y  +416.328, Z    +0.000, E1  +404.105, E3 -194863.172}
SPL {X  -159.990, Y  +459.824, Z    +0.000, E1  +420.326, E3 -194883.093}
SPL {X  -159.990, Y  +561.459, Z    +0.000, E1  +423.923, E3 -194961.960}
SPL {X  -159.990, Y  +574.787, Z    +0.000, E1  +423.950, E3 -194975.756}
SPL {X  -159.990, Y  +590.041, Z    +0.000, E1  +423.939, E3 -194991.617}
SPL {X  -159.990, Y  +601.352, Z    +0.000, E1  +423.918, E3 -195003.403}
SPL {X  -159.990, Y  +614.998, Z    +0.000, E1  +423.962, E3 -195017.488}
SPL {X  -159.990, Y  +632.576, Z    +0.000, E1  +423.953, E3 -195035.753}
SPL {X  -159.990, Y  +648.849, Z    +0.000, E1  +423.945, E3 -195052.682}
SPL {X  -159.990, Y  +661.195, Z    +0.000, E1  +423.915, E3 -195065.583}
SPL {X  -159.965, Y  +674.349, Z    +0.000, E1  +423.939, E3 -195079.219}
SPL {X  -159.404, Y  +685.179, Z    +0.000, E1  +423.831, E3 -195091.098}
SPL {X  -158.535, Y  +693.032, Z    +0.000, E1  +423.713, E3 -195100.148}
SPL {X  -156.949, Y  +702.544, Z    +0.000, E1  +423.501, E3 -195111.653}
SPL {X  -154.903, Y  +711.525, Z    +0.000, E1  +423.186, E3 -195123.124}
SPL {X  -153.138, Y  +717.820, Z    +0.000, E1  +422.909, E3 -195131.479}
SPL {X  -151.229, Y  +723.716, Z    +0.000, E1  +422.630, E3 -195139.489}
SPL {X  -149.219, Y  +729.211, Z    +0.000, E1  +422.307, E3 -195147.197}
SPL {X  -146.537, Y  +735.716, Z    +0.000, E1  +421.906, E3 -195156.540}
SPL {X  -143.476, Y  +742.291, Z    +0.000, E1  +421.379, E3 -195166.300}
SPL {X  -141.015, Y  +747.074, Z    +0.000, E1  +420.958, E3 -195173.556}
SPL {X  -137.271, Y  +753.679, Z    +0.000, E1  +420.346, E3 -195183.695}
SPL {X  -133.306, Y  +759.967, Z    +0.000, E1  +419.584, E3 -195193.646}
SPL {X  -112.019, Y  +785.730, Z    +0.000, E1  +410.795, E3 -195296.387}
ENDSPLINE

SPLINE
SPL {X  -138.335, Y  +751.876, Z    +0.000, E1  +401.001, E3 -195410.686}
SPL {X  -150.285, Y  +726.376, Z    +0.000, E1  +392.667, E3 -195429.095}
SPL {X  -154.601, Y  +712.673, Z    +0.000, E1  +386.751, E3 -195434.700}
SPL {X  -158.303, Y  +694.673, Z    +0.000, E1  +377.238, E3 -195439.369}
SPL {X  -159.774, Y  +679.819, Z    +0.000, E1  +367.840, E3 -195441.443}
SPL {X  -159.990, Y  +671.106, Z    +0.000, E1  +361.459, E3 -195441.964}
SPL {X  -159.990, Y  +668.525, Z    +0.000, E1  +359.125, E3 -195442.009}
SPL {X  -159.990, Y  +664.817, Z    +0.000, E1  +353.836, E3 -195442.150}
SPL {X  -159.990, Y  +661.286, Z    +0.000, E1  +348.294, E3 -195442.412}
SPL {X  -159.990, Y  +654.198, Z    +0.000, E1  +336.753, E3 -195443.323}
SPL {X  -159.990, Y  +643.777, Z    +0.000, E1  +322.140, E3 -195445.488}
SPL {X  -159.990, Y  +634.027, Z    +0.000, E1  +313.116, E3 -195448.400}
SPL {X  -159.990, Y  +589.014, Z    +0.000, E1  +298.500, E3 -195468.451}
SPL {X  -159.990, Y  +484.717, Z    +0.000, E1  +295.169, E3 -195546.634}
SPL {X  -159.990, Y  +469.712, Z    +0.000, E1  +295.152, E3 -195561.572}
SPL {X  -159.990, Y  +456.089, Z    +0.000, E1  +295.174, E3 -195575.187}
SPL {X  -159.990, Y  +443.816, Z    +0.000, E1  +295.158, E3 -195587.388}
SPL {X  -159.990, Y  +410.689, Z    +0.000, E1  +292.263, E3 -195595.112}
SPL {X  -159.990, Y  +399.563, Z    +0.000, E1  +292.427, E3 -195606.351}
SPL {X  -159.990, Y  +393.786, Z    +0.000, E1  +293.391, E3 -195619.339}
SPL {X  -159.990, Y  +387.038, Z    +0.000, E1  +293.844, E3 -195629.195}
SPL {X  -159.983, Y  +380.995, Z    +0.000, E1  +294.559, E3 -195640.764}
SPL {X  -159.795, Y  +374.602, Z    +0.000, E1  +295.796, E3 -195656.783}
SPL {X  -159.306, Y  +367.719, Z    +0.000, E1  +296.544, E3 -195669.240}
SPL {X  -158.431, Y  +360.219, Z    +0.000, E1  +296.670, E3 -195678.091}
SPL {X  -156.653, Y  +349.995, Z    +0.000, E1  +296.892, E3 -195690.660}
SPL {X  -153.792, Y  +338.401, Z    +0.000, E1  +297.323, E3 -195705.829}
SPL {X  -151.244, Y  +330.327, Z    +0.000, E1  +297.748, E3 -195716.982}
SPL {X  -148.909, Y  +323.994, Z    +0.000, E1  +298.107, E3 -195725.968}
SPL {X  -146.667, Y  +318.581, Z    +0.000, E1  +298.485, E3 -195733.888}
SPL {X  -144.416, Y  +313.647, Z    +0.000, E1  +298.845, E3 -195741.224}
SPL {X  -141.484, Y  +307.808, Z    +0.000, E1  +299.342, E3 -195750.117}
SPL {X  -139.055, Y  +303.377, Z    +0.000, E1  +299.788, E3 -195757.029}
SPL {X  -136.464, Y  +298.988, Z    +0.000, E1  +300.231, E3 -195763.904}
SPL {X  -133.486, Y  +294.305, Z    +0.000, E1  +300.785, E3 -195771.366}
SPL {X  -111.268, Y  +267.538, Z    +0.000, E1  +309.436, E3 -195879.265}
ENDSPLINE

SPLINE
SPL {X  -140.331, Y  +305.662, Z    +0.000, E1  +319.927, E3 -195991.333}
SPL {X  -153.176, Y  +336.305, Z    +0.000, E1  +330.872, E3 -196009.887}
SPL {X  -158.263, Y  +359.056, Z    +0.000, E1  +342.551, E3 -196016.562}
SPL {X  -159.616, Y  +371.564, Z    +0.000, E1  +350.434, E3 -196018.467}
SPL {X  -159.946, Y  +378.747, Z    +0.000, E1  +355.440, E3 -196019.062}
SPL {X  -159.990, Y  +384.172, Z    +0.000, E1  +359.586, E3 -196019.241}
SPL {X  -159.990, Y  +385.853, Z    +0.000, E1  +361.539, E3 -196019.265}
SPL {X  -159.990, Y  +389.234, Z    +0.000, E1  +366.142, E3 -196019.410}
SPL {X  -159.990, Y  +395.814, Z    +0.000, E1  +376.762, E3 -196020.011}
SPL {X  -159.990, Y  +404.858, Z    +0.000, E1  +391.125, E3 -196021.525}
SPL {X  -159.990, Y  +416.328, Z    +0.000, E1  +404.105, E3 -196024.462}
SPL {X  -159.990, Y  +459.824, Z    +0.000, E1  +420.326, E3 -196044.384}
SPL {X  -159.990, Y  +565.974, Z    +0.000, E1  +423.959, E3 -196127.873}
SPL {X  -159.990, Y  +578.588, Z    +0.000, E1  +423.918, E3 -196141.052}
SPL {X  -159.990, Y  +590.041, Z    +0.000, E1  +423.939, E3 -196152.907}
SPL {X  -159.990, Y  +601.352, Z    +0.000, E1  +423.918, E3 -196164.693}
SPL {X  -159.990, Y  +610.973, Z    +0.000, E1  +423.927, E3 -196174.661}
SPL {X  -159.990, Y  +624.756, Z    +0.000, E1  +423.949, E3 -196188.939}
SPL {X  -159.990, Y  +636.914, Z    +0.000, E1  +423.917, E3 -196201.615}
SPL {X  -159.990, Y  +648.849, Z    +0.000, E1  +423.945, E3 -196213.972}
SPL {X  -159.990, Y  +661.195, Z    +0.000, E1  +423.915, E3 -196226.873}
SPL {X  -159.990, Y  +670.369, Z    +0.000, E1  +423.912, E3 -196236.406}
SPL {X  -159.643, Y  +682.032, Z    +0.000, E1  +423.894, E3 -196248.821}
SPL {X  -158.070, Y  +696.212, Z    +0.000, E1  +423.682, E3 -196265.159}
SPL {X  -155.481, Y  +709.215, Z    +0.000, E1  +423.310, E3 -196281.351}
SPL {X  -153.138, Y  +717.820, Z    +0.000, E1  +422.909, E3 -196292.769}
SPL {X  -151.229, Y  +723.716, Z    +0.000, E1  +422.630, E3 -196300.779}
SPL {X  -149.219, Y  +729.211, Z    +0.000, E1  +422.307, E3 -196308.487}
SPL {X  -146.537, Y  +735.716, Z    +0.000, E1  +421.906, E3 -196317.830}
SPL {X  -143.476, Y  +742.291, Z    +0.000, E1  +421.379, E3 -196327.590}
SPL {X  -141.015, Y  +747.074, Z    +0.000, E1  +420.958, E3 -196334.847}
SPL {X  -138.539, Y  +751.523, Z    +0.000, E1  +420.526, E3 -196341.681}
SPL {X  -136.299, Y  +755.281, Z    +0.000, E1  +420.128, E3 -196347.543}
SPL {X  -133.306, Y  +759.967, Z    +0.000, E1  +419.584, E3 -196354.937}
SPL {X  -112.019, Y  +785.730, Z    +0.000, E1  +410.795, E3 -196457.677}
ENDSPLINE

SPLINE
SPL {X  -126.527, Y  +769.417, Z    +0.000, E1  +405.012, E3 -196547.530}
SPL {X  -141.954, Y  +745.296, Z    +0.000, E1  +399.179, E3 -196578.728}
SPL {X  -153.384, Y  +716.997, Z    +0.000, E1  +388.774, E3 -196594.347}
SPL {X  -158.303, Y  +694.673, Z    +0.000, E1  +377.238, E3 -196600.659}
SPL {X  -159.604, Y  +682.609, Z    +0.000, E1  +369.664, E3 -196602.469}
SPL {X  -159.964, Y  +674.389, Z    +0.000, E1  +363.956, E3 -196603.131}
SPL {X  -159.990, Y  +669.409, Z    +0.000, E1  +360.015, E3 -196603.284}
SPL {X  -159.990, Y  +667.272, Z    +0.000, E1  +357.329, E3 -196603.327}
SPL {X  -159.990, Y  +664.817, Z    +0.000, E1  +353.836, E3 -196603.440}
SPL {X  -159.990, Y  +661.286, Z    +0.000, E1  +348.294, E3 -196603.702}
SPL {X  -159.990, Y  +654.198, Z    +0.000, E1  +336.753, E3 -196604.613}
SPL {X  -159.990, Y  +640.109, Z    +0.000, E1  +318.471, E3 -196607.876}
SPL {X  -159.990, Y  +589.014, Z    +0.000, E1  +298.500, E3 -196629.742}
SPL {X  -159.990, Y  +484.717, Z    +0.000, E1  +295.169, E3 -196707.925}
SPL {X  -159.990, Y  +469.712, Z    +0.000, E1  +295.152, E3 -196722.862}
SPL {X  -159.990, Y  +456.089, Z    +0.000, E1  +295.174, E3 -196736.478}
SPL {X  -159.990, Y  +443.816, Z    +0.000, E1  +295.158, E3 -196748.678}
SPL {X  -159.990, Y  +405.035, Z    +0.000, E1  +292.209, E3 -196760.949}
SPL {X  -159.990, Y  +395.217, Z    +0.000, E1  +293.078, E3 -196777.057}
SPL {X  -159.990, Y  +385.177, Z    +0.000, E1  +294.011, E3 -196793.746}
SPL {X  -159.935, Y  +378.300, Z    +0.000, E1  +295.100, E3 -196808.956}
SPL {X  -159.533, Y  +370.414, Z    +0.000, E1  +296.253, E3 -196825.865}
SPL {X  -158.431, Y  +360.219, Z    +0.000, E1  +296.670, E3 -196839.382}
SPL {X  -157.299, Y  +353.279, Z    +0.000, E1  +296.835, E3 -196847.878}
SPL {X  -155.242, Y  +343.812, Z    +0.000, E1  +297.102, E3 -196859.926}
SPL {X  -151.999, Y  +332.569, Z    +0.000, E1  +297.592, E3 -196875.085}
SPL {X  -148.909, Y  +323.994, Z    +0.000, E1  +298.107, E3 -196887.258}
SPL {X  -146.667, Y  +318.581, Z    +0.000, E1  +298.485, E3 -196895.178}
SPL {X  -144.416, Y  +313.647, Z    +0.000, E1  +298.845, E3 -196902.515}
SPL {X  -141.484, Y  +307.808, Z    +0.000, E1  +299.342, E3 -196911.408}
SPL {X  -139.055, Y  +303.377, Z    +0.000, E1  +299.788, E3 -196918.320}
SPL {X  -136.464, Y  +298.988, Z    +0.000, E1  +300.231, E3 -196925.194}
SPL {X  -133.486, Y  +294.305, Z    +0.000, E1  +300.785, E3 -196932.656}
SPL {X  -111.268, Y  +267.538, Z    +0.000, E1  +309.436, E3 -197040.555}
ENDSPLINE

SPLINE
SPL {X  -140.331, Y  +305.662, Z    +0.000, E1  +319.927, E3 -197152.623}
SPL {X  -153.176, Y  +336.305, Z    +0.000, E1  +330.872, E3 -197171.178}
SPL {X  -158.263, Y  +359.056, Z    +0.000, E1  +342.551, E3 -197177.852}
SPL {X  -159.616, Y  +371.564, Z    +0.000, E1  +350.434, E3 -197179.757}
SPL {X  -159.946, Y  +378.747, Z    +0.000, E1  +355.440, E3 -197180.352}
SPL {X  -159.990, Y  +384.172, Z    +0.000, E1  +359.586, E3 -197180.531}
SPL {X  -159.990, Y  +386.890, Z    +0.000, E1  +362.742, E3 -197180.592}
SPL {X  -159.990, Y  +392.248, Z    +0.000, E1  +370.895, E3 -197180.920}
SPL {X  -159.990, Y  +398.030, Z    +0.000, E1  +380.706, E3 -197181.571}
SPL {X  -159.990, Y  +404.858, Z    +0.000, E1  +391.125, E3 -197182.815}
SPL {X  -159.990, Y  +416.328, Z    +0.000, E1  +404.105, E3 -197185.752}
SPL {X  -159.990, Y  +459.824, Z    +0.000, E1  +420.326, E3 -197205.674}
SPL {X  -159.990, Y  +565.974, Z    +0.000, E1  +423.959, E3 -197289.163}
SPL {X  -159.990, Y  +578.588, Z    +0.000, E1  +423.918, E3 -197302.342}
SPL {X  -159.990, Y  +590.041, Z    +0.000, E1  +423.939, E3 -197314.197}
SPL {X  -159.990, Y  +601.352, Z    +0.000, E1  +423.918, E3 -197325.983}
SPL {X  -159.990, Y  +610.973, Z    +0.000, E1  +423.927, E3 -197335.952}
SPL {X  -159.990, Y  +624.756, Z    +0.000, E1  +423.949, E3 -197350.229}
SPL {X  -159.990, Y  +640.674, Z    +0.000, E1  +423.943, E3 -197366.766}
SPL {X  -159.990, Y  +652.355, Z    +0.000, E1  +423.915, E3 -197378.965}
SPL {X  -159.990, Y  +665.748, Z    +0.000, E1  +423.953, E3 -197392.819}
SPL {X  -159.643, Y  +682.032, Z    +0.000, E1  +423.894, E3 -197410.112}
SPL {X  -158.070, Y  +696.212, Z    +0.000, E1  +423.682, E3 -197426.450}
SPL {X  -155.481, Y  +709.215, Z    +0.000, E1  +423.310, E3 -197442.641}
SPL {X  -153.138, Y  +717.820, Z    +0.000, E1  +422.909, E3 -197454.059}
SPL {X  -151.229, Y  +723.716, Z    +0.000, E1  +422.630, E3 -197462.069}
SPL {X  -149.219, Y  +729.211, Z    +0.000, E1  +422.307, E3 -197469.777}
SPL {X  -146.537, Y  +735.716, Z    +0.000, E1  +421.906, E3 -197479.121}
SPL {X  -143.476, Y  +742.291, Z    +0.000, E1  +421.379, E3 -197488.881}
SPL {X  -141.015, Y  +747.074, Z    +0.000, E1  +420.958, E3 -197496.137}
SPL {X  -137.271, Y  +753.679, Z    +0.000, E1  +420.346, E3 -197506.275}
SPL {X  -133.306, Y  +759.967, Z    +0.000, E1  +419.584, E3 -197516.227}
SPL {X  -112.019, Y  +785.730, Z    +0.000, E1  +410.795, E3 -197618.968}
ENDSPLINE

SPLINE
SPL {X  -138.335, Y  +751.876, Z    +0.000, E1  +401.001, E3 -197733.266}
SPL {X  -150.285, Y  +726.376, Z    +0.000, E1  +392.667, E3 -197751.676}
SPL {X  -156.272, Y  +705.789, Z    +0.000, E1  +383.396, E3 -197759.312}
SPL {X  -159.413, Y  +685.076, Z    +0.000, E1  +371.341, E3 -197763.450}
SPL {X  -159.964, Y  +674.389, Z    +0.000, E1  +363.956, E3 -197764.421}
SPL {X  -159.990, Y  +670.214, Z    +0.000, E1  +360.653, E3 -197764.567}
SPL {X  -159.990, Y  +669.154, Z    +0.000, E1  +359.694, E3 -197764.576}
SPL {X  -159.990, Y  +666.004, Z    +0.000, E1  +355.742, E3 -197764.676}
SPL {X  -159.990, Y  +661.286, Z    +0.000, E1  +348.294, E3 -197764.992}
SPL {X  -159.990, Y  +656.470, Z    +0.000, E1  +340.220, E3 -197765.530}
SPL {X  -159.990, Y  +651.555, Z    +0.000, E1  +332.416, E3 -197766.338}
SPL {X  -159.990, Y  +640.109, Z    +0.000, E1  +318.471, E3 -197769.166}
SPL {X  -159.990, Y  +589.014, Z    +0.000, E1  +298.500, E3 -197791.032}
SPL {X  -159.990, Y  +484.717, Z    +0.000, E1  +295.169, E3 -197869.215}
SPL {X  -159.990, Y  +469.712, Z    +0.000, E1  +295.152, E3 -197884.152}
SPL {X  -159.990, Y  +456.089, Z    +0.000, E1  +295.174, E3 -197897.768}
SPL {X  -159.990, Y  +443.816, Z    +0.000, E1  +295.158, E3 -197909.968}
SPL {X  -159.990, Y  +405.035, Z    +0.000, E1  +292.209, E3 -197922.239}
SPL {X  -159.990, Y  +397.824, Z    +0.000, E1  +292.709, E3 -197932.601}
SPL {X  -159.990, Y  +393.786, Z    +0.000, E1  +293.391, E3 -197941.920}
SPL {X  -159.990, Y  +385.177, Z    +0.000, E1  +294.011, E3 -197955.036}
SPL {X  -159.935, Y  +378.300, Z    +0.000, E1  +295.100, E3 -197970.246}
SPL {X  -159.716, Y  +373.142, Z    +0.000, E1  +296.084, E3 -197982.787}
SPL {X  -158.852, Y  +363.449, Z    +0.000, E1  +296.568, E3 -197996.737}
SPL {X  -157.299, Y  +353.279, Z    +0.000, E1  +296.835, E3 -198009.169}
SPL {X  -155.242, Y  +343.812, Z    +0.000, E1  +297.102, E3 -198021.217}
SPL {X  -151.999, Y  +332.569, Z    +0.000, E1  +297.592, E3 -198036.375}
SPL {X  -148.909, Y  +323.994, Z    +0.000, E1  +298.107, E3 -198048.548}
SPL {X  -146.667, Y  +318.581, Z    +0.000, E1  +298.485, E3 -198056.469}
SPL {X  -144.416, Y  +313.647, Z    +0.000, E1  +298.845, E3 -198063.805}
SPL {X  -141.484, Y  +307.808, Z    +0.000, E1  +299.342, E3 -198072.698}
SPL {X  -139.055, Y  +303.377, Z    +0.000, E1  +299.788, E3 -198079.610}
SPL {X  -136.464, Y  +298.988, Z    +0.000, E1  +300.231, E3 -198086.485}
SPL {X  -133.486, Y  +294.305, Z    +0.000, E1  +300.785, E3 -198093.947}
SPL {X  -111.268, Y  +267.538, Z    +0.000, E1  +309.436, E3 -198201.846}
ENDSPLINE

SPLINE
SPL {X  -140.331, Y  +305.662, Z    +0.000, E1  +319.927, E3 -198313.914}
SPL {X  -153.176, Y  +336.305, Z    +0.000, E1  +330.872, E3 -198332.468}
SPL {X  -158.263, Y  +359.056, Z    +0.000, E1  +342.551, E3 -198339.143}
SPL {X  -159.616, Y  +371.564, Z    +0.000, E1  +350.434, E3 -198341.048}
SPL {X  -159.946, Y  +378.747, Z    +0.000, E1  +355.440, E3 -198341.643}
SPL {X  -159.990, Y  +384.172, Z    +0.000, E1  +359.586, E3 -198341.821}
SPL {X  -159.990, Y  +385.853, Z    +0.000, E1  +361.539, E3 -198341.846}
SPL {X  -159.990, Y  +389.234, Z    +0.000, E1  +366.142, E3 -198341.991}
SPL {X  -159.990, Y  +395.814, Z    +0.000, E1  +376.762, E3 -198342.592}
SPL {X  -159.990, Y  +404.858, Z    +0.000, E1  +391.125, E3 -198344.106}
SPL {X  -159.990, Y  +416.328, Z    +0.000, E1  +404.105, E3 -198347.042}
SPL {X  -159.990, Y  +459.824, Z    +0.000, E1  +420.326, E3 -198366.964}
SPL {X  -159.990, Y  +565.974, Z    +0.000, E1  +423.959, E3 -198450.453}
SPL {X  -159.990, Y  +578.588, Z    +0.000, E1  +423.918, E3 -198463.633}
SPL {X  -159.990, Y  +590.041, Z    +0.000, E1  +423.939, E3 -198475.487}
SPL {X  -159.990, Y  +601.352, Z    +0.000, E1  +423.918, E3 -198487.274}
SPL {X  -159.990, Y  +610.973, Z    +0.000, E1  +423.927, E3 -198497.242}
SPL {X  -159.990, Y  +624.756, Z    +0.000, E1  +423.949, E3 -198511.520}
SPL {X  -159.990, Y  +636.914, Z    +0.000, E1  +423.917, E3 -198524.196}
SPL {X  -159.990, Y  +648.849, Z    +0.000, E1  +423.945, E3 -198536.553}
SPL {X  -159.990, Y  +661.195, Z    +0.000, E1  +423.915, E3 -198549.454}
SPL {X  -159.965, Y  +674.349, Z    +0.000, E1  +423.939, E3 -198563.090}
SPL {X  -159.404, Y  +685.179, Z    +0.000, E1  +423.831, E3 -198574.969}
SPL {X  -158.535, Y  +693.032, Z    +0.000, E1  +423.713, E3 -198584.019}
SPL {X  -156.949, Y  +702.544, Z    +0.000, E1  +423.501, E3 -198595.524}
SPL {X  -154.903, Y  +711.525, Z    +0.000, E1  +423.186, E3 -198606.995}
SPL {X  -153.138, Y  +717.820, Z    +0.000, E1  +422.909, E3 -198615.350}
SPL {X  -151.229, Y  +723.716, Z    +0.000, E1  +422.630, E3 -198623.360}
SPL {X  -149.219, Y  +729.211, Z    +0.000, E1  +422.307, E3 -198631.068}
SPL {X  -146.537, Y  +735.716, Z    +0.000, E1  +421.906, E3 -198640.411}
SPL {X  -143.476, Y  +742.291, Z    +0.000, E1  +421.379, E3 -198650.171}
SPL {X  -141.015, Y  +747.074, Z    +0.000, E1  +420.958, E3 -198657.427}
SPL {X  -137.271, Y  +753.679, Z    +0.000, E1  +420.346, E3 -198667.566}
SPL {X  -133.306, Y  +759.967, Z    +0.000, E1  +419.584, E3 -198677.517}
SPL {X  -112.019, Y  +785.730, Z    +0.000, E1  +410.795, E3 -198780.258}
ENDSPLINE

SPLINE
SPL {X  -138.335, Y  +751.876, Z    +0.000, E1  +401.001, E3 -198894.557}
SPL {X  -150.285, Y  +726.376, Z    +0.000, E1  +392.667, E3 -198912.966}
SPL {X  -156.272, Y  +705.789, Z    +0.000, E1  +383.396, E3 -198920.602}
SPL {X  -159.413, Y  +685.076, Z    +0.000, E1  +371.341, E3 -198924.741}
SPL {X  -159.964, Y  +674.389, Z    +0.000, E1  +363.956, E3 -198925.711}
SPL {X  -159.990, Y  +669.409, Z    +0.000, E1  +360.015, E3 -198925.864}
SPL {X  -159.990, Y  +667.272, Z    +0.000, E1  +357.329, E3 -198925.908}
SPL {X  -159.990, Y  +664.817, Z    +0.000, E1  +353.836, E3 -198926.021}
SPL {X  -159.990, Y  +661.286, Z    +0.000, E1  +348.294, E3 -198926.283}
SPL {X  -159.990, Y  +654.198, Z    +0.000, E1  +336.753, E3 -198927.194}
SPL {X  -159.990, Y  +640.109, Z    +0.000, E1  +318.471, E3 -198930.457}
SPL {X  -159.990, Y  +589.014, Z    +0.000, E1  +298.500, E3 -198952.322}
SPL {X  -159.990, Y  +484.717, Z    +0.000, E1  +295.169, E3 -199030.505}
SPL {X  -159.990, Y  +474.300, Z    +0.000, E1  +295.184, E3 -199040.933}
SPL {X  -159.990, Y  +465.825, Z    +0.000, E1  +295.182, E3 -199049.373}
SPL {X  -159.990, Y  +451.559, Z    +0.000, E1  +295.138, E3 -199063.510}
SPL {X  -159.990, Y  +438.393, Z    +0.000, E1  +295.184, E3 -199076.731}
SPL {X  -159.990, Y  +405.035, Z    +0.000, E1  +292.209, E3 -199083.529}
SPL {X  -159.990, Y  +395.217, Z    +0.000, E1  +293.078, E3 -199099.638}
SPL {X  -159.990, Y  +387.038, Z    +0.000, E1  +293.844, E3 -199113.066}
SPL {X  -159.983, Y  +380.995, Z    +0.000, E1  +294.559, E3 -199124.635}
SPL {X  -159.795, Y  +374.602, Z    +0.000, E1  +295.796, E3 -199140.654}
SPL {X  -158.852, Y  +363.449, Z    +0.000, E1  +296.568, E3 -199158.027}
SPL {X  -156.653, Y  +349.995, Z    +0.000, E1  +296.892, E3 -199174.531}
SPL {X  -153.792, Y  +338.401, Z    +0.000, E1  +297.323, E3 -199189.700}
SPL {X  -151.244, Y  +330.327, Z    +0.000, E1  +297.748, E3 -199200.853}
SPL {X  -148.909, Y  +323.994, Z    +0.000, E1  +298.107, E3 -199209.839}
SPL {X  -146.667, Y  +318.581, Z    +0.000, E1  +298.485, E3 -199217.759}
SPL {X  -144.416, Y  +313.647, Z    +0.000, E1  +298.845, E3 -199225.095}
SPL {X  -141.484, Y  +307.808, Z    +0.000, E1  +299.342, E3 -199233.988}
SPL {X  -139.055, Y  +303.377, Z    +0.000, E1  +299.788, E3 -199240.900}
SPL {X  -136.464, Y  +298.988, Z    +0.000, E1  +300.231, E3 -199247.775}
SPL {X  -133.486, Y  +294.305, Z    +0.000, E1  +300.785, E3 -199255.237}
SPL {X  -111.268, Y  +267.538, Z    +0.000, E1  +309.436, E3 -199363.136}
ENDSPLINE

SPLINE
SPL {X  -140.331, Y  +305.662, Z    +0.000, E1  +319.927, E3 -199475.204}
SPL {X  -153.176, Y  +336.305, Z    +0.000, E1  +330.872, E3 -199493.758}
SPL {X  -157.724, Y  +355.668, Z    +0.000, E1  +340.639, E3 -199499.767}
SPL {X  -159.465, Y  +369.545, Z    +0.000, E1  +349.053, E3 -199502.089}
SPL {X  -159.983, Y  +381.031, Z    +0.000, E1  +357.053, E3 -199503.029}
SPL {X  -159.990, Y  +384.524, Z    +0.000, E1  +359.995, E3 -199503.117}
SPL {X  -159.990, Y  +386.890, Z    +0.000, E1  +362.742, E3 -199503.173}
SPL {X  -159.990, Y  +392.248, Z    +0.000, E1  +370.895, E3 -199503.500}
SPL {X  -159.990, Y  +398.030, Z    +0.000, E1  +380.706, E3 -199504.152}
SPL {X  -159.990, Y  +404.858, Z    +0.000, E1  +391.125, E3 -199505.396}
SPL {X  -159.990, Y  +416.328, Z    +0.000, E1  +404.105, E3 -199508.333}
SPL {X  -159.990, Y  +459.824, Z    +0.000, E1  +420.326, E3 -199528.255}
SPL {X  -159.990, Y  +565.974, Z    +0.000, E1  +423.959, E3 -199611.744}
SPL {X  -159.990, Y  +578.588, Z    +0.000, E1  +423.918, E3 -199624.923}
SPL {X  -159.990, Y  +590.041, Z    +0.000, E1  +423.939, E3 -199636.778}
SPL {X  -159.990, Y  +601.352, Z    +0.000, E1  +423.918, E3 -199648.564}
SPL {X  -159.990, Y  +614.998, Z    +0.000, E1  +423.962, E3 -199662.649}
SPL {X  -159.990, Y  +628.256, Z    +0.000, E1  +423.919, E3 -199676.498}
SPL {X  -159.990, Y  +640.674, Z    +0.000, E1  +423.943, E3 -199689.347}
SPL {X  -159.990, Y  +657.298, Z    +0.000, E1  +423.953, E3 -199706.619}
SPL {X  -159.990, Y  +670.369, Z    +0.000, E1  +423.912, E3 -199720.276}
SPL {X  -159.643, Y  +682.032, Z    +0.000, E1  +423.894, E3 -199732.692}
SPL {X  -158.070, Y  +696.212, Z    +0.000, E1  +423.682, E3 -199749.030}
SPL {X  -155.481, Y  +709.215, Z    +0.000, E1  +423.310, E3 -199765.221}
SPL {X  -153.138, Y  +717.820, Z    +0.000, E1  +422.909, E3 -199776.640}
SPL {X  -151.229, Y  +723.716, Z    +0.000, E1  +422.630, E3 -199784.650}
SPL {X  -149.219, Y  +729.211, Z    +0.000, E1  +422.307, E3 -199792.358}
SPL {X  -146.537, Y  +735.716, Z    +0.000, E1  +421.906, E3 -199801.701}
SPL {X  -143.476, Y  +742.291, Z    +0.000, E1  +421.379, E3 -199811.461}
SPL {X  -141.015, Y  +747.074, Z    +0.000, E1  +420.958, E3 -199818.718}
SPL {X  -137.271, Y  +753.679, Z    +0.000, E1  +420.346, E3 -199828.856}
SPL {X  -133.306, Y  +759.967, Z    +0.000, E1  +419.584, E3 -199838.808}
SPL {X  -112.019, Y  +785.730, Z    +0.000, E1  +410.795, E3 -199941.548}
ENDSPLINE

SPLINE
SPL {X  -126.527, Y  +769.417, Z    +0.000, E1  +405.012, E3 -200031.401}
SPL {X  -141.954, Y  +745.296, Z    +0.000, E1  +399.179, E3 -200062.599}
SPL {X  -153.384, Y  +716.997, Z    +0.000, E1  +388.774, E3 -200078.218}
SPL {X  -158.303, Y  +694.673, Z    +0.000, E1  +377.238, E3 -200084.530}
SPL {X  -159.604, Y  +682.609, Z    +0.000, E1  +369.664, E3 -200086.340}
SPL {X  -159.964, Y  +674.389, Z    +0.000, E1  +363.956, E3 -200087.002}
SPL {X  -159.990, Y  +669.409, Z    +0.000, E1  +360.015, E3 -200087.155}
SPL {X  -159.990, Y  +666.004, Z    +0.000, E1  +355.742, E3 -200087.256}
SPL {X  -159.990, Y  +661.286, Z    +0.000, E1  +348.294, E3 -200087.573}
SPL {X  -159.990, Y  +654.198, Z    +0.000, E1  +336.753, E3 -200088.484}
SPL {X  -159.990, Y  +640.109, Z    +0.000, E1  +318.471, E3 -200091.747}
SPL {X  -159.990, Y  +589.014, Z    +0.000, E1  +298.500, E3 -200113.613}
SPL {X  -159.990, Y  +484.717, Z    +0.000, E1  +295.169, E3 -200191.796}
SPL {X  -159.990, Y  +474.300, Z    +0.000, E1  +295.184, E3 -200202.224}
SPL {X  -159.990, Y  +465.825, Z    +0.000, E1  +295.182, E3 -200210.663}
SPL {X  -159.990, Y  +451.559, Z    +0.000, E1  +295.138, E3 -200224.800}
SPL {X  -159.990, Y  +423.512, Z    +0.000, E1  +293.559, E3 -200239.234}
SPL {X  -159.990, Y  +399.563, Z    +0.000, E1  +292.427, E3 -200251.512}
SPL {X  -159.990, Y  +393.786, Z    +0.000, E1  +293.391, E3 -200264.501}
SPL {X  -159.990, Y  +387.038, Z    +0.000, E1  +293.844, E3 -200274.356}
SPL {X  -159.983, Y  +380.995, Z    +0.000, E1  +294.559, E3 -200285.925}
SPL {X  -159.898, Y  +377.064, Z    +0.000, E1  +295.481, E3 -200296.739}
SPL {X  -159.716, Y  +373.142, Z    +0.000, E1  +296.084, E3 -200305.368}
SPL {X  -158.852, Y  +363.449, Z    +0.000, E1  +296.568, E3 -200319.317}
SPL {X  -157.299, Y  +353.279, Z    +0.000, E1  +296.835, E3 -200331.749}
SPL {X  -155.242, Y  +343.812, Z    +0.000, E1  +297.102, E3 -200343.797}
SPL {X  -151.999, Y  +332.569, Z    +0.000, E1  +297.592, E3 -200358.956}
SPL {X  -148.909, Y  +323.994, Z    +0.000, E1  +298.107, E3 -200371.129}
SPL {X  -146.667, Y  +318.581, Z    +0.000, E1  +298.485, E3 -200379.049}
SPL {X  -144.416, Y  +313.647, Z    +0.000, E1  +298.845, E3 -200386.386}
SPL {X  -141.484, Y  +307.808, Z    +0.000, E1  +299.342, E3 -200395.279}
SPL {X  -139.055, Y  +303.377, Z    +0.000, E1  +299.788, E3 -200402.191}
SPL {X  -136.464, Y  +298.988, Z    +0.000, E1  +300.231, E3 -200409.065}
SPL {X  -133.486, Y  +294.305, Z    +0.000, E1  +300.785, E3 -200416.527}
SPL {X  -111.268, Y  +267.538, Z    +0.000, E1  +309.436, E3 -200524.426}
ENDSPLINE

SPLINE
SPL {X  -140.331, Y  +305.662, Z    +0.000, E1  +319.927, E3 -200636.494}
SPL {X  -153.176, Y  +336.305, Z    +0.000, E1  +330.872, E3 -200655.049}
SPL {X  -158.263, Y  +359.056, Z    +0.000, E1  +342.551, E3 -200661.723}
SPL {X  -159.616, Y  +371.564, Z    +0.000, E1  +350.434, E3 -200663.628}
SPL {X  -159.983, Y  +381.031, Z    +0.000, E1  +357.053, E3 -200664.319}
SPL {X  -159.990, Y  +385.049, Z    +0.000, E1  +360.437, E3 -200664.415}
SPL {X  -159.990, Y  +389.234, Z    +0.000, E1  +366.142, E3 -200664.571}
SPL {X  -159.990, Y  +395.814, Z    +0.000, E1  +376.762, E3 -200665.172}
SPL {X  -159.990, Y  +404.858, Z    +0.000, E1  +391.125, E3 -200666.686}
SPL {X  -159.990, Y  +416.328, Z    +0.000, E1  +404.105, E3 -200669.623}
SPL {X  -159.990, Y  +459.824, Z    +0.000, E1  +420.326, E3 -200689.545}
SPL {X  -159.990, Y  +565.974, Z    +0.000, E1  +423.959, E3 -200773.034}
SPL {X  -159.990, Y  +582.903, Z    +0.000, E1  +423.951, E3 -200790.631}
SPL {X  -159.990, Y  +598.374, Z    +0.000, E1  +423.941, E3 -200806.717}
SPL {X  -159.990, Y  +614.998, Z    +0.000, E1  +423.962, E3 -200823.939}
SPL {X  -159.990, Y  +632.576, Z    +0.000, E1  +423.953, E3 -200842.205}
SPL {X  -159.990, Y  +648.849, Z    +0.000, E1  +423.945, E3 -200859.134}
SPL {X  -159.990, Y  +665.748, Z    +0.000, E1  +423.953, E3 -200876.690}
SPL {X  -159.643, Y  +682.032, Z    +0.000, E1  +423.894, E3 -200893.983}
SPL {X  -158.070, Y  +696.212, Z    +0.000, E1  +423.682, E3 -200910.321}
SPL {X  -155.481, Y  +709.215, Z    +0.000, E1  +423.310, E3 -200926.512}
SPL {X  -153.138, Y  +717.820, Z    +0.000, E1  +422.909, E3 -200937.930}
SPL {X  -151.229, Y  +723.716, Z    +0.000, E1  +422.630, E3 -200945.940}
SPL {X  -148.422, Y  +731.231, Z    +0.000, E1  +422.207, E3 -200956.498}
SPL {X  -145.802, Y  +737.367, Z    +0.000, E1  +421.758, E3 -200965.451}
SPL {X  -143.476, Y  +742.291, Z    +0.000, E1  +421.379, E3 -200972.751}
SPL {X  -141.015, Y  +747.074, Z    +0.000, E1  +420.958, E3 -200980.008}
SPL {X  -138.539, Y  +751.523, Z    +0.000, E1  +420.526, E3 -200986.843}
SPL {X  -136.299, Y  +755.281, Z    +0.000, E1  +420.128, E3 -200992.704}
SPL {X  -133.306, Y  +759.967, Z    +0.000, E1  +419.584, E3 -201000.098}
SPL {X  -112.019, Y  +785.730, Z    +0.000, E1  +410.795, E3 -201102.839}
ENDSPLINE

SPLINE
SPL {X  -138.335, Y  +751.876, Z    +0.000, E1  +401.001, E3 -201217.137}
SPL {X  -150.285, Y  +726.376, Z    +0.000, E1  +392.667, E3 -201235.547}
SPL {X  -154.601, Y  +712.673, Z    +0.000, E1  +386.751, E3 -201241.152}
SPL {X  -158.303, Y  +694.673, Z    +0.000, E1  +377.238, E3 -201245.821}
SPL {X  -159.774, Y  +679.819, Z    +0.000, E1  +367.840, E3 -201247.895}
SPL {X  -159.990, Y  +671.106, Z    +0.000, E1  +361.459, E3 -201248.416}
SPL {X  -159.990, Y  +669.154, Z    +0.000, E1  +359.694, E3 -201248.447}
SPL {X  -159.990, Y  +666.004, Z    +0.000, E1  +355.742, E3 -201248.547}
SPL {X  -159.990, Y  +661.286, Z    +0.000, E1  +348.294, E3 -201248.863}
SPL {X  -159.990, Y  +656.470, Z    +0.000, E1  +340.220, E3 -201249.401}
SPL {X  -159.990, Y  +651.555, Z    +0.000, E1  +332.416, E3 -201250.208}
SPL {X  -159.990, Y  +640.109, Z    +0.000, E1  +318.471, E3 -201253.037}
SPL {X  -159.990, Y  +589.014, Z    +0.000, E1  +298.500, E3 -201274.903}
SPL {X  -159.990, Y  +484.717, Z    +0.000, E1  +295.169, E3 -201353.086}
SPL {X  -159.990, Y  +469.712, Z    +0.000, E1  +295.152, E3 -201368.023}
SPL {X  -159.990, Y  +456.089, Z    +0.000, E1  +295.174, E3 -201381.639}
SPL {X  -159.990, Y  +443.816, Z    +0.000, E1  +295.158, E3 -201393.839}
SPL {X  -159.990, Y  +405.035, Z    +0.000, E1  +292.209, E3 -201406.110}
SPL {X  -159.990, Y  +395.217, Z    +0.000, E1  +293.078, E3 -201422.218}
SPL {X  -159.990, Y  +387.038, Z    +0.000, E1  +293.844, E3 -201435.647}
SPL {X  -159.983, Y  +380.995, Z    +0.000, E1  +294.559, E3 -201447.215}
SPL {X  -159.795, Y  +374.602, Z    +0.000, E1  +295.796, E3 -201463.235}
SPL {X  -158.852, Y  +363.449, Z    +0.000, E1  +296.568, E3 -201480.608}
SPL {X  -156.653, Y  +349.995, Z    +0.000, E1  +296.892, E3 -201497.111}
SPL {X  -153.792, Y  +338.401, Z    +0.000, E1  +297.323, E3 -201512.281}
SPL {X  -151.244, Y  +330.327, Z    +0.000, E1  +297.748, E3 -201523.434}
SPL {X  -148.909, Y  +323.994, Z    +0.000, E1  +298.107, E3 -201532.419}
SPL {X  -146.667, Y  +318.581, Z    +0.000, E1  +298.485, E3 -201540.340}
SPL {X  -144.416, Y  +313.647, Z    +0.000, E1  +298.845, E3 -201547.676}
SPL {X  -141.484, Y  +307.808, Z    +0.000, E1  +299.342, E3 -201556.569}
SPL {X  -139.055, Y  +303.377, Z    +0.000, E1  +299.788, E3 -201563.481}
SPL {X  -136.464, Y  +298.988, Z    +0.000, E1  +300.231, E3 -201570.356}
SPL {X  -133.486, Y  +294.305, Z    +0.000, E1  +300.785, E3 -201577.818}
SPL {X  -111.268, Y  +267.538, Z    +0.000, E1  +309.436, E3 -201685.717}
ENDSPLINE

SPLINE
SPL {X  -140.331, Y  +305.662, Z    +0.000, E1  +319.927, E3 -201797.785}
SPL {X  -153.176, Y  +336.305, Z    +0.000, E1  +330.872, E3 -201816.339}
SPL {X  -158.263, Y  +359.056, Z    +0.000, E1  +342.551, E3 -201823.014}
SPL {X  -159.616, Y  +371.564, Z    +0.000, E1  +350.434, E3 -201824.919}
SPL {X  -159.983, Y  +381.031, Z    +0.000, E1  +357.053, E3 -201825.609}
SPL {X  -159.990, Y  +385.049, Z    +0.000, E1  +360.437, E3 -201825.705}
SPL {X  -159.990, Y  +389.234, Z    +0.000, E1  +366.142, E3 -201825.862}
SPL {X  -159.990, Y  +395.814, Z    +0.000, E1  +376.762, E3 -201826.463}
SPL {X  -159.990, Y  +404.858, Z    +0.000, E1  +391.125, E3 -201827.977}
SPL {X  -159.990, Y  +416.328, Z    +0.000, E1  +404.105, E3 -201830.913}
SPL {X  -159.990, Y  +459.824, Z    +0.000, E1  +420.326, E3 -201850.835}
SPL {X  -159.990, Y  +565.974, Z    +0.000, E1  +423.959, E3 -201934.324}
SPL {X  -159.990, Y  +582.903, Z    +0.000, E1  +423.951, E3 -201951.921}
SPL {X  -159.990, Y  +598.374, Z    +0.000, E1  +423.941, E3 -201968.008}
SPL {X  -159.990, Y  +614.998, Z    +0.000, E1  +423.962, E3 -201985.230}
SPL {X  -159.990, Y  +632.576, Z    +0.000, E1  +423.953, E3 -202003.495}
SPL {X  -159.990, Y  +648.849, Z    +0.000, E1  +423.945, E3 -202020.424}
SPL {X  -159.990, Y  +665.748, Z    +0.000, E1  +423.953, E3 -202037.980}
SPL {X  -159.643, Y  +682.032, Z    +0.000, E1  +423.894, E3 -202055.273}
SPL {X  -158.070, Y  +696.212, Z    +0.000, E1  +423.682, E3 -202071.611}
SPL {X  -155.481, Y  +709.215, Z    +0.000, E1  +423.310, E3 -202087.802}
SPL {X  -153.138, Y  +717.820, Z    +0.000, E1  +422.909, E3 -202099.221}
SPL {X  -151.229, Y  +723.716, Z    +0.000, E1  +422.630, E3 -202107.231}
SPL {X  -148.422, Y  +731.231, Z    +0.000, E1  +422.207, E3 -202117.788}
SPL {X  -145.802, Y  +737.367, Z    +0.000, E1  +421.758, E3 -202126.741}
SPL {X  -143.476, Y  +742.291, Z    +0.000, E1  +421.379, E3 -202134.042}
SPL {X  -141.015, Y  +747.074, Z    +0.000, E1  +420.958, E3 -202141.298}
SPL {X  -138.539, Y  +751.523, Z    +0.000, E1  +420.526, E3 -202148.133}
SPL {X  -136.299, Y  +755.281, Z    +0.000, E1  +420.128, E3 -202153.994}
SPL {X  -133.306, Y  +759.967, Z    +0.000, E1  +419.584, E3 -202161.388}
SPL {X  -112.019, Y  +785.730, Z    +0.000, E1  +410.795, E3 -202264.129}
ENDSPLINE

SPLINE
SPL {X  -126.527, Y  +769.417, Z    +0.000, E1  +405.012, E3 -202353.982}
SPL {X  -145.458, Y  +738.125, Z    +0.000, E1  +396.959, E3 -202390.064}
SPL {X  -156.272, Y  +705.789, Z    +0.000, E1  +383.396, E3 -202404.473}
SPL {X  -159.413, Y  +685.076, Z    +0.000, E1  +371.341, E3 -202408.612}
SPL {X  -159.901, Y  +676.826, Z    +0.000, E1  +365.664, E3 -202409.444}
SPL {X  -159.990, Y  +671.106, Z    +0.000, E1  +361.459, E3 -202409.706}
SPL {X  -159.990, Y  +668.525, Z    +0.000, E1  +359.125, E3 -202409.751}
SPL {X  -159.990, Y  +664.817, Z    +0.000, E1  +353.836, E3 -202409.892}
SPL {X  -159.990, Y  +661.286, Z    +0.000, E1  +348.294, E3 -202410.153}
SPL {X  -159.990, Y  +654.198, Z    +0.000, E1  +336.753, E3 -202411.065}
SPL {X  -159.990, Y  +640.109, Z    +0.000, E1  +318.471, E3 -202414.328}
SPL {X  -159.990, Y  +589.014, Z    +0.000, E1  +298.500, E3 -202436.193}
SPL {X  -159.990, Y  +484.717, Z    +0.000, E1  +295.169, E3 -202514.376}
SPL {X  -159.990, Y  +469.712, Z    +0.000, E1  +295.152, E3 -202529.314}
SPL {X  -159.990, Y  +456.089, Z    +0.000, E1  +295.174, E3 -202542.929}
SPL {X  -159.990, Y  +443.816, Z    +0.000, E1  +295.158, E3 -202555.129}
SPL {X  -159.990, Y  +405.035, Z    +0.000, E1  +292.209, E3 -202567.400}
SPL {X  -159.990, Y  +395.217, Z    +0.000, E1  +293.078, E3 -202583.509}
SPL {X  -159.990, Y  +385.177, Z    +0.000, E1  +294.011, E3 -202600.198}
SPL {X  -159.935, Y  +378.300, Z    +0.000, E1  +295.100, E3 -202615.408}
SPL {X  -159.533, Y  +370.414, Z    +0.000, E1  +296.253, E3 -202632.317}
SPL {X  -158.431, Y  +360.219, Z    +0.000, E1  +296.670, E3 -202645.833}
SPL {X  -157.299, Y  +353.279, Z    +0.000, E1  +296.835, E3 -202654.330}
SPL {X  -155.242, Y  +343.812, Z    +0.000, E1  +297.102, E3 -202666.378}
SPL {X  -151.999, Y  +332.569, Z    +0.000, E1  +297.592, E3 -202681.536}
SPL {X  -148.909, Y  +323.994, Z    +0.000, E1  +298.107, E3 -202693.710}
SPL {X  -146.667, Y  +318.581, Z    +0.000, E1  +298.485, E3 -202701.630}
SPL {X  -144.416, Y  +313.647, Z    +0.000, E1  +298.845, E3 -202708.966}
SPL {X  -141.484, Y  +307.808, Z    +0.000, E1  +299.342, E3 -202717.859}
SPL {X  -139.055, Y  +303.377, Z    +0.000, E1  +299.788, E3 -202724.771}
SPL {X  -136.464, Y  +298.988, Z    +0.000, E1  +300.231, E3 -202731.646}
SPL {X  -133.486, Y  +294.305, Z    +0.000, E1  +300.785, E3 -202739.108}
SPL {X  -111.268, Y  +267.538, Z    +0.000, E1  +309.436, E3 -202847.007}
ENDSPLINE

SPLINE
SPL {X  -140.331, Y  +305.662, Z    +0.000, E1  +319.927, E3 -202959.075}
SPL {X  -153.176, Y  +336.305, Z    +0.000, E1  +330.872, E3 -202977.629}
SPL {X  -157.724, Y  +355.668, Z    +0.000, E1  +340.639, E3 -202983.637}
SPL {X  -159.465, Y  +369.545, Z    +0.000, E1  +349.053, E3 -202985.960}
SPL {X  -159.983, Y  +381.031, Z    +0.000, E1  +357.053, E3 -202986.900}
SPL {X  -159.990, Y  +384.524, Z    +0.000, E1  +359.995, E3 -202986.988}
SPL {X  -159.990, Y  +386.890, Z    +0.000, E1  +362.742, E3 -202987.044}
SPL {X  -159.990, Y  +392.248, Z    +0.000, E1  +370.895, E3 -202987.371}
SPL {X  -159.990, Y  +398.030, Z    +0.000, E1  +380.706, E3 -202988.023}
SPL {X  -159.990, Y  +404.858, Z    +0.000, E1  +391.125, E3 -202989.267}
SPL {X  -159.990, Y  +416.328, Z    +0.000, E1  +404.105, E3 -202992.204}
SPL {X  -159.990, Y  +459.824, Z    +0.000, E1  +420.326, E3 -203012.126}
SPL {X  -159.990, Y  +565.974, Z    +0.000, E1  +423.959, E3 -203095.615}
SPL {X  -159.990, Y  +578.588, Z    +0.000, E1  +423.918, E3 -203108.794}
SPL {X  -159.990, Y  +590.041, Z    +0.000, E1  +423.939, E3 -203120.649}
SPL {X  -159.990, Y  +601.352, Z    +0.000, E1  +423.918, E3 -203132.435}
SPL {X  -159.990, Y  +614.998, Z    +0.000, E1  +423.962, E3 -203146.520}
SPL {X  -159.990, Y  +628.256, Z    +0.000, E1  +423.919, E3 -203160.368}
SPL {X  -159.990, Y  +640.674, Z    +0.000, E1  +423.943, E3 -203173.218}
SPL {X  -159.990, Y  +657.298, Z    +0.000, E1  +423.953, E3 -203190.490}
SPL {X  -159.990, Y  +670.369, Z    +0.000, E1  +423.912, E3 -203204.147}
SPL {X  -159.643, Y  +682.032, Z    +0.000, E1  +423.894, E3 -203216.563}
SPL {X  -158.070, Y  +696.212, Z    +0.000, E1  +423.682, E3 -203232.901}
SPL {X  -155.481, Y  +709.215, Z    +0.000, E1  +423.310, E3 -203249.092}
SPL {X  -153.138, Y  +717.820, Z    +0.000, E1  +422.909, E3 -203260.511}
SPL {X  -151.229, Y  +723.716, Z    +0.000, E1  +422.630, E3 -203268.521}
SPL {X  -149.219, Y  +729.211, Z    +0.000, E1  +422.307, E3 -203276.229}
SPL {X  -146.537, Y  +735.716, Z    +0.000, E1  +421.906, E3 -203285.572}
SPL {X  -143.476, Y  +742.291, Z    +0.000, E1  +421.379, E3 -203295.332}
SPL {X  -141.015, Y  +747.074, Z    +0.000, E1  +420.958, E3 -203302.589}
SPL {X  -137.271, Y  +753.679, Z    +0.000, E1  +420.346, E3 -203312.727}
SPL {X  -133.306, Y  +759.967, Z    +0.000, E1  +419.584, E3 -203322.679}
SPL {X  -112.019, Y  +785.730, Z    +0.000, E1  +410.795, E3 -203425.419}
ENDSPLINE

SPLINE
SPL {X  -126.527, Y  +769.417, Z    +0.000, E1  +405.012, E3 -203515.272}
SPL {X  -141.954, Y  +745.296, Z    +0.000, E1  +399.179, E3 -203546.470}
SPL {X  -153.384, Y  +716.997, Z    +0.000, E1  +388.774, E3 -203562.089}
SPL {X  -158.303, Y  +694.673, Z    +0.000, E1  +377.238, E3 -203568.401}
SPL {X  -159.604, Y  +682.609, Z    +0.000, E1  +369.664, E3 -203570.211}
SPL {X  -159.964, Y  +674.389, Z    +0.000, E1  +363.956, E3 -203570.873}
SPL {X  -159.990, Y  +669.409, Z    +0.000, E1  +360.015, E3 -203571.026}
SPL {X  -159.990, Y  +666.004, Z    +0.000, E1  +355.742, E3 -203571.127}
SPL {X  -159.990, Y  +661.286, Z    +0.000, E1  +348.294, E3 -203571.444}
SPL {X  -159.990, Y  +654.198, Z    +0.000, E1  +336.753, E3 -203572.355}
SPL {X  -159.990, Y  +640.109, Z    +0.000, E1  +318.471, E3 -203575.618}
SPL {X  -159.990, Y  +589.014, Z    +0.000, E1  +298.500, E3 -203597.484}
SPL {X  -159.990, Y  +484.717, Z    +0.000, E1  +295.169, E3 -203675.667}
SPL {X  -159.990, Y  +474.300, Z    +0.000, E1  +295.184, E3 -203686.095}
SPL {X  -159.990, Y  +465.825, Z    +0.000, E1  +295.182, E3 -203694.534}
SPL {X  -159.990, Y  +451.559, Z    +0.000, E1  +295.138, E3 -203708.671}
SPL {X  -159.990, Y  +423.512, Z    +0.000, E1  +293.559, E3 -203723.105}
SPL {X  -159.990, Y  +399.563, Z    +0.000, E1  +292.427, E3 -203735.383}
SPL {X  -159.990, Y  +393.786, Z    +0.000, E1  +293.391, E3 -203748.372}
SPL {X  -159.990, Y  +387.038, Z    +0.000, E1  +293.844, E3 -203758.227}
SPL {X  -159.983, Y  +380.995, Z    +0.000, E1  +294.559, E3 -203769.796}
SPL {X  -159.898, Y  +377.064, Z    +0.000, E1  +295.481, E3 -203780.610}
SPL {X  -159.716, Y  +373.142, Z    +0.000, E1  +296.084, E3 -203789.239}
SPL {X  -158.852, Y  +363.449, Z    +0.000, E1  +296.568, E3 -203803.188}
SPL {X  -157.299, Y  +353.279, Z    +0.000, E1  +296.835, E3 -203815.620}
SPL {X  -155.242, Y  +343.812, Z    +0.000, E1  +297.102, E3 -203827.668}
SPL {X  -151.999, Y  +332.569, Z    +0.000, E1  +297.592, E3 -203842.826}
SPL {X  -148.909, Y  +323.994, Z    +0.000, E1  +298.107, E3 -203855.000}
SPL {X  -146.667, Y  +318.581, Z    +0.000, E1  +298.485, E3 -203862.920}
SPL {X  -144.416, Y  +313.647, Z    +0.000, E1  +298.845, E3 -203870.256}
SPL {X  -141.484, Y  +307.808, Z    +0.000, E1  +299.342, E3 -203879.150}
SPL {X  -139.055, Y  +303.377, Z    +0.000, E1  +299.788, E3 -203886.062}
SPL {X  -136.464, Y  +298.988, Z    +0.000, E1  +300.231, E3 -203892.936}
SPL {X  -133.486, Y  +294.305, Z    +0.000, E1  +300.785, E3 -203900.398}
SPL {X  -111.268, Y  +267.538, Z    +0.000, E1  +309.436, E3 -204008.297}
ENDSPLINE

SPLINE
SPL {X  -140.331, Y  +305.662, Z    +0.000, E1  +319.927, E3 -204120.365}
SPL {X  -153.176, Y  +336.305, Z    +0.000, E1  +330.872, E3 -204138.920}
SPL {X  -158.263, Y  +359.056, Z    +0.000, E1  +342.551, E3 -204145.594}
SPL {X  -159.616, Y  +371.564, Z    +0.000, E1  +350.434, E3 -204147.499}
SPL {X  -159.983, Y  +381.031, Z    +0.000, E1  +357.053, E3 -204148.190}
SPL {X  -159.990, Y  +385.049, Z    +0.000, E1  +360.437, E3 -204148.286}
SPL {X  -159.990, Y  +389.234, Z    +0.000, E1  +366.142, E3 -204148.442}
SPL {X  -159.990, Y  +395.814, Z    +0.000, E1  +376.762, E3 -204149.043}
SPL {X  -159.990, Y  +404.858, Z    +0.000, E1  +391.125, E3 -204150.557}
SPL {X  -159.990, Y  +416.328, Z    +0.000, E1  +404.105, E3 -204153.494}
SPL {X  -159.990, Y  +459.824, Z    +0.000, E1  +420.326, E3 -204173.416}
SPL {X  -159.990, Y  +565.974, Z    +0.000, E1  +423.959, E3 -204256.905}
SPL {X  -159.990, Y  +578.588, Z    +0.000, E1  +423.918, E3 -204270.084}
SPL {X  -159.990, Y  +590.041, Z    +0.000, E1  +423.939, E3 -204281.939}
SPL {X  -159.990, Y  +601.352, Z    +0.000, E1  +423.918, E3 -204293.725}
SPL {X  -159.990, Y  +610.973, Z    +0.000, E1  +423.927, E3 -204303.694}
SPL {X  -159.990, Y  +624.756, Z    +0.000, E1  +423.949, E3 -204317.971}
SPL {X  -159.990, Y  +640.674, Z    +0.000, E1  +423.943, E3 -204334.508}
SPL {X  -159.990, Y  +657.298, Z    +0.000, E1  +423.953, E3 -204351.780}
SPL {X  -159.965, Y  +674.349, Z    +0.000, E1  +423.939, E3 -204369.542}
SPL {X  -159.404, Y  +685.179, Z    +0.000, E1  +423.831, E3 -204381.421}
SPL {X  -158.535, Y  +693.032, Z    +0.000, E1  +423.713, E3 -204390.471}
SPL {X  -156.949, Y  +702.544, Z    +0.000, E1  +423.501, E3 -204401.976}
SPL {X  -154.903, Y  +711.525, Z    +0.000, E1  +423.186, E3 -204413.447}
SPL {X  -153.138, Y  +717.820, Z    +0.000, E1  +422.909, E3 -204421.801}
SPL {X  -151.229, Y  +723.716, Z    +0.000, E1  +422.630, E3 -204429.811}
SPL {X  -149.219, Y  +729.211, Z    +0.000, E1  +422.307, E3 -204437.519}
SPL {X  -146.537, Y  +735.716, Z    +0.000, E1  +421.906, E3 -204446.862}
SPL {X  -143.476, Y  +742.291, Z    +0.000, E1  +421.379, E3 -204456.622}
SPL {X  -141.015, Y  +747.074, Z    +0.000, E1  +420.958, E3 -204463.879}
SPL {X  -138.539, Y  +751.523, Z    +0.000, E1  +420.526, E3 -204470.714}
SPL {X  -136.299, Y  +755.281, Z    +0.000, E1  +420.128, E3 -204476.575}
SPL {X  -133.306, Y  +759.967, Z    +0.000, E1  +419.584, E3 -204483.969}
SPL {X  -112.019, Y  +785.730, Z    +0.000, E1  +410.795, E3 -204586.710}
ENDSPLINE

SPLINE
SPL {X  -138.335, Y  +751.876, Z    +0.000, E1  +401.001, E3 -204701.008}
SPL {X  -153.384, Y  +716.997, Z    +0.000, E1  +388.774, E3 -204723.380}
SPL {X  -157.578, Y  +699.176, Z    +0.000, E1  +379.774, E3 -204728.809}
SPL {X  -159.413, Y  +685.076, Z    +0.000, E1  +371.341, E3 -204731.192}
SPL {X  -159.901, Y  +676.826, Z    +0.000, E1  +365.664, E3 -204732.025}
SPL {X  -159.990, Y  +671.106, Z    +0.000, E1  +361.459, E3 -204732.287}
SPL {X  -159.990, Y  +669.154, Z    +0.000, E1  +359.694, E3 -204732.318}
SPL {X  -159.990, Y  +666.004, Z    +0.000, E1  +355.742, E3 -204732.418}
SPL {X  -159.990, Y  +661.286, Z    +0.000, E1  +348.294, E3 -204732.734}
SPL {X  -159.990, Y  +654.198, Z    +0.000, E1  +336.753, E3 -204733.645}
SPL {X  -159.990, Y  +640.109, Z    +0.000, E1  +318.471, E3 -204736.908}
SPL {X  -159.990, Y  +589.014, Z    +0.000, E1  +298.500, E3 -204758.774}
SPL {X  -159.990, Y  +484.717, Z    +0.000, E1  +295.169, E3 -204836.957}
SPL {X  -159.990, Y  +469.712, Z    +0.000, E1  +295.152, E3 -204851.894}
SPL {X  -159.990, Y  +451.559, Z    +0.000, E1  +295.138, E3 -204869.961}
SPL {X  -159.990, Y  +423.512, Z    +0.000, E1  +293.559, E3 -204884.395}
SPL {X  -159.990, Y  +399.563, Z    +0.000, E1  +292.427, E3 -204896.674}
SPL {X  -159.990, Y  +393.786, Z    +0.000, E1  +293.391, E3 -204909.662}
SPL {X  -159.990, Y  +387.038, Z    +0.000, E1  +293.844, E3 -204919.518}
SPL {X  -159.983, Y  +380.995, Z    +0.000, E1  +294.559, E3 -204931.086}
SPL {X  -159.795, Y  +374.602, Z    +0.000, E1  +295.796, E3 -204947.106}
SPL {X  -159.306, Y  +367.719, Z    +0.000, E1  +296.544, E3 -204959.563}
SPL {X  -158.431, Y  +360.219, Z    +0.000, E1  +296.670, E3 -204968.414}
SPL {X  -157.299, Y  +353.279, Z    +0.000, E1  +296.835, E3 -204976.911}
SPL {X  -155.242, Y  +343.812, Z    +0.000, E1  +297.102, E3 -204988.959}
SPL {X  -151.999, Y  +332.569, Z    +0.000, E1  +297.592, E3 -205004.117}
SPL {X  -148.909, Y  +323.994, Z    +0.000, E1  +298.107, E3 -205016.290}
SPL {X  -146.667, Y  +318.581, Z    +0.000, E1  +298.485, E3 -205024.211}
SPL {X  -144.416, Y  +313.647, Z    +0.000, E1  +298.845, E3 -205031.547}
SPL {X  -141.484, Y  +307.808, Z    +0.000, E1  +299.342, E3 -205040.440}
SPL {X  -139.055, Y  +303.377, Z    +0.000, E1  +299.788, E3 -205047.352}
SPL {X  -136.464, Y  +298.988, Z    +0.000, E1  +300.231, E3 -205054.226}
SPL {X  -133.486, Y  +294.305, Z    +0.000, E1  +300.785, E3 -205061.689}
SPL {X  -111.268, Y  +267.538, Z    +0.000, E1  +309.436, E3 -205169.588}
ENDSPLINE

SPLINE
SPL {X  -140.331, Y  +305.662, Z    +0.000, E1  +319.927, E3 -205281.656}
SPL {X  -153.176, Y  +336.305, Z    +0.000, E1  +330.872, E3 -205300.210}
SPL {X  -157.724, Y  +355.668, Z    +0.000, E1  +340.639, E3 -205306.218}
SPL {X  -159.465, Y  +369.545, Z    +0.000, E1  +349.053, E3 -205308.541}
SPL {X  -159.983, Y  +381.031, Z    +0.000, E1  +357.053, E3 -205309.480}
SPL {X  -159.990, Y  +384.524, Z    +0.000, E1  +359.995, E3 -205309.568}
SPL {X  -159.990, Y  +386.890, Z    +0.000, E1  +362.742, E3 -205309.624}
SPL {X  -159.990, Y  +392.248, Z    +0.000, E1  +370.895, E3 -205309.952}
SPL {X  -159.990, Y  +398.030, Z    +0.000, E1  +380.706, E3 -205310.603}
SPL {X  -159.990, Y  +404.858, Z    +0.000, E1  +391.125, E3 -205311.848}
SPL {X  -159.990, Y  +416.328, Z    +0.000, E1  +404.105, E3 -205314.784}
SPL {X  -159.990, Y  +459.824, Z    +0.000, E1  +420.326, E3 -205334.706}
SPL {X  -159.990, Y  +561.459, Z    +0.000, E1  +423.923, E3 -205413.573}
SPL {X  -159.990, Y  +574.787, Z    +0.000, E1  +423.950, E3 -205427.369}
SPL {X  -159.990, Y  +590.041, Z    +0.000, E1  +423.939, E3 -205443.229}
SPL {X  -159.990, Y  +601.352, Z    +0.000, E1  +423.918, E3 -205455.016}
SPL {X  -159.990, Y  +610.973, Z    +0.000, E1  +423.927, E3 -205464.984}
SPL {X  -159.990, Y  +624.756, Z    +0.000, E1  +423.949, E3 -205479.262}
SPL {X  -159.990, Y  +640.674, Z    +0.000, E1  +423.943, E3 -205495.798}
SPL {X  -159.990, Y  +652.355, Z    +0.000, E1  +423.915, E3 -205507.997}
SPL {X  -159.990, Y  +661.195, Z    +0.000, E1  +423.915, E3 -205517.196}
SPL {X  -159.965, Y  +674.349, Z    +0.000, E1  +423.939, E3 -205530.832}
SPL {X  -159.404, Y  +685.179, Z    +0.000, E1  +423.831, E3 -205542.711}
SPL {X  -158.535, Y  +693.032, Z    +0.000, E1  +423.713, E3 -205551.761}
SPL {X  -156.949, Y  +702.544, Z    +0.000, E1  +423.501, E3 -205563.266}
SPL {X  -154.903, Y  +711.525, Z    +0.000, E1  +423.186, E3 -205574.737}
SPL {X  -153.138, Y  +717.820, Z    +0.000, E1  +422.909, E3 -205583.092}
SPL {X  -151.229, Y  +723.716, Z    +0.000, E1  +422.630, E3 -205591.101}
SPL {X  -149.219, Y  +729.211, Z    +0.000, E1  +422.307, E3 -205598.810}
SPL {X  -146.537, Y  +735.716, Z    +0.000, E1  +421.906, E3 -205608.153}
SPL {X  -143.476, Y  +742.291, Z    +0.000, E1  +421.379, E3 -205617.913}
SPL {X  -141.015, Y  +747.074, Z    +0.000, E1  +420.958, E3 -205625.169}
SPL {X  -138.539, Y  +751.523, Z    +0.000, E1  +420.526, E3 -205632.004}
SPL {X  -136.299, Y  +755.281, Z    +0.000, E1  +420.128, E3 -205637.865}
SPL {X  -133.306, Y  +759.967, Z    +0.000, E1  +419.584, E3 -205645.259}
SPL {X  -112.019, Y  +785.730, Z    +0.000, E1  +410.795, E3 -205748.000}
ENDSPLINE

